KUKA KRL program: MyProgram_129().src

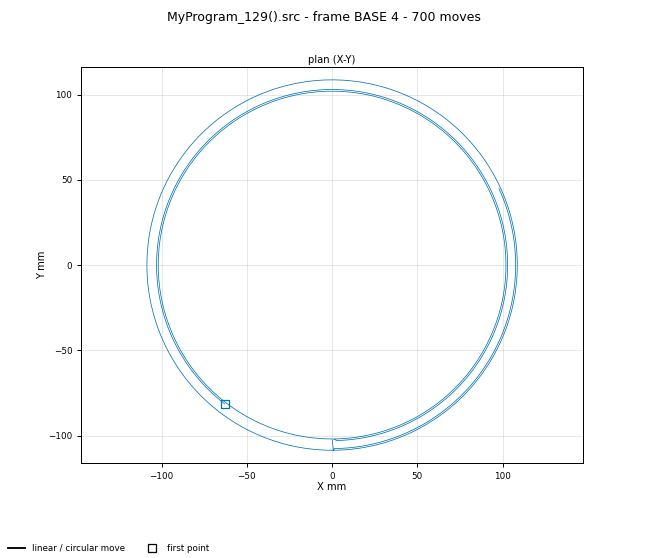
[picture p0: tool path of MyProgram_129().src in frame BASE 4, 700 of 700 moves have a stored position in this frame; points joined in program order, loops and branches not executed]
&ACCESS RVP
&REL 1
&PARAM TEMPLATE = C:\KRC\Roboter\Template\vorgabe
&PARAM EDITMASK = *
DEF MyProgram_129()
; ---- Setting reference (Base) ----
$BASE = BASE_DATA[4]

; --------------------------
; ---- Setting tool (TCP) ----
$TOOL = TOOL_DATA[3]
; --------------------------

$VEL.CP = VEL_APROX_PRINT
Startdeposition()
$VEL.CP = VEL_PRINT
LIN {X -62.9658,Y -81.4453,Z 106,A -132.2913,B 24.9442,C -1.7248,E1 24.9012,E2 217.9169} C_DIS
LIN {X -65.6067,Y -79.3337,Z 106,A -134.1331,B 24.9439,C -1.7297,E1 24.8972,E2 219.7539} C_DIS
LIN {X -68.2811,Y -77.0452,Z 106,A -136.1102,B 24.9437,C -1.7329,E1 24.893,E2 221.7312} C_DIS
LIN {X -70.4655,Y -75.0509,Z 106,A -137.9265,B 24.9439,C -1.7301,E1 24.8893,E2 223.5615} C_DIS
LIN {X -73.3174,Y -72.2675,Z 106,A -139.9622,B 24.9432,C -1.7414,E1 24.8853,E2 225.5791} C_DIS
LIN {X -75.616,Y -69.8596,Z 106,A -142.0598,B 24.9435,C -1.7367,E1 24.8812,E2 227.697} C_DIS
LIN {X -78.3073,Y -66.8281,Z 106,A -144.1543,B 24.9428,C -1.7476,E1 24.8774,E2 229.7748} C_DIS
LIN {X -80.8839,Y -63.6856,Z 106,A -146.4557,B 24.9425,C -1.7516,E1 24.8734,E2 232.0776} C_DIS
LIN {X -82.6713,Y -61.3501,Z 106,A -147.9403,B 24.9419,C -1.7609,E1 24.8709,E2 233.547} C_DIS
LIN {X -84.3493,Y -59.0196,Z 106,A -149.6735,B 24.9419,C -1.7602,E1 24.8681,E2 235.2905} C_DIS
LIN {X -86.3097,Y -56.1161,Z 106,A -151.7179,B 24.9419,C -1.7618,E1 24.8649,E2 237.3412} C_DIS
LIN {X -88.3102,Y -52.9122,Z 106,A -153.6162,B 24.941,C -1.7746,E1 24.8622,E2 239.2189} C_DIS
LIN {X -89.3427,Y -51.1462,Z 106,A -155.0866,B 24.9415,C -1.766,E1 24.8601,E2 240.7174} C_DIS
LIN {X -91.3359,Y -47.498,Z 106,A -157.1631,B 24.9406,C -1.7806,E1 24.8574,E2 242.77} C_DIS
LIN {X -93.0269,Y -44.0942,Z 106,A -159.4092,B 24.9405,C -1.782,E1 24.8547,E2 245.025} C_DIS
LIN {X -94.4755,Y -40.8958,Z 106,A -161.3998,B 24.9402,C -1.7863,E1 24.8524,E2 247.0162} C_DIS
LIN {X -95.9861,Y -37.2142,Z 106,A -163.4255,B 24.9393,C -1.7994,E1 24.8503,E2 249.0222} C_DIS
LIN {X -97.1234,Y -34.133,Z 106,A -165.4942,B 24.9395,C -1.7964,E1 24.8484,E2 251.1096} C_DIS
LIN {X -98.3351,Y -30.4667,Z 106,A -167.5356,B 24.9388,C -1.8066,E1 24.8466,E2 253.1384} C_DIS
LIN {X -99.2194,Y -27.4578,Z 106,A -169.3316,B 24.9386,C -1.8101,E1 24.8453,E2 254.9364} C_DIS
LIN {X -100.529,Y -22.1809,Z 106,A -172.0309,B 24.9372,C -1.8308,E1 24.8435,E2 257.6021} C_DIS
LIN {X -101.1949,Y -18.9188,Z 106,A -174.3718,B 24.9379,C -1.8197,E1 24.8422,E2 259.9835} C_DIS
LIN {X -101.8925,Y -14.6964,Z 106,A -176.5465,B 24.9369,C -1.8344,E1 24.8413,E2 262.136} C_DIS
LIN {X -102.234,Y -12.0934,Z 106,A -178.0467,B 24.9367,C -1.8377,E1 24.8408,E2 263.6374} C_DIS
LIN {X -102.5546,Y -8.9886,Z 106,A -179.9416,B 24.9367,C -1.8377,E1 24.8403,E2 265.5434} C_DIS
LIN {X -102.8206,Y -5.1232,Z 106,A 177.9162,B 24.9362,C -1.8452,E1 24.8399,E2 267.6808} C_DIS
LIN {X -102.9266,Y -2.0367,Z 106,A 176.3907,B 24.9353,C -1.8574,E1 24.8399,E2 269.1864} C_DIS
LIN {X -102.9421,Y 1.0814,Z 106,A 174.6385,B 24.935,C -1.8624,E1 24.8399,E2 270.9372} C_DIS
LIN {X -102.8555,Y 4.3316,Z 106,A 172.9749,B 24.9342,C -1.8733,E1 24.8399,E2 272.5849} C_DIS
LIN {X -102.6601,Y 7.6926,Z 106,A 170.758,B 24.9346,C -1.8675,E1 24.8404,E2 274.8289} C_DIS
LIN {X -102.3213,Y 11.3472,Z 106,A 168.6519,B 24.9343,C -1.8719,E1 24.8409,E2 276.9371} C_DIS
LIN {X -101.8299,Y 15.1348,Z 106,A 166.6862,B 24.9334,C -1.8843,E1 24.8417,E2 278.8851} C_DIS
LIN {X -101.2979,Y 18.3511,Z 106,A 164.7721,B 24.9333,C -1.8867,E1 24.8426,E2 280.8047} C_DIS
LIN {X -100.3856,Y 22.8227,Z 106,A 162.208,B 24.9328,C -1.894,E1 24.8441,E2 283.3665} C_DIS
LIN {X -99.542,Y 26.2634,Z 106,A 160.1806,B 24.9324,C -1.8983,E1 24.8455,E2 285.3955} C_DIS
LIN {X -98.7388,Y 29.1324,Z 106,A 158.4759,B 24.9322,C -1.902,E1 24.8468,E2 287.1013} C_DIS
LIN {X -97.7556,Y 32.2837,Z 106,A 156.7577,B 24.9315,C -1.9118,E1 24.8483,E2 288.8059} C_DIS
LIN {X -96.565,Y 35.6848,Z 106,A 154.8063,B 24.9309,C -1.9199,E1 24.8501,E2 290.7491} C_DIS
LIN {X -95.1884,Y 39.2093,Z 106,A 152.6847,B 24.9305,C -1.9258,E1 24.8523,E2 292.8684} C_DIS
LIN {X -93.4142,Y 43.2647,Z 106,A 150.4424,B 24.9294,C -1.9409,E1 24.8548,E2 295.0869} C_DIS
LIN {X -92.6832,Y 44.8096,Z 106,A 148.8667,B 24.9307,C -1.9222,E1 24.8568,E2 296.7159} C_DIS
LIN {X -90.7079,Y 48.6857,Z 106,A 146.6291,B 24.9298,C -1.9357,E1 24.8596,E2 298.9333} C_DIS
LIN {X -88.9696,Y 51.7954,Z 106,A 144.6192,B 24.9294,C -1.9405,E1 24.8624,E2 300.9422} C_DIS
LIN {X -87.387,Y 54.4202,Z 106,A 142.3126,B 24.9306,C -1.9247,E1 24.8659,E2 303.2983} C_DIS
LIN {X -84.9704,Y 58.1231,Z 106,A 140.4496,B 24.9286,C -1.9521,E1 24.8687,E2 305.1051} C_DIS
LIN {X -82.9524,Y 60.9668,Z 106,A 138.6482,B 24.9278,C -1.9623,E1 24.8716,E2 306.8911} C_DIS
LIN {X -80.8826,Y 63.6871,Z 106,A 136.6902,B 24.9276,C -1.9654,E1 24.875,E2 308.8509} C_DIS
LIN {X -78.8684,Y 66.1667,Z 106,A 134.7875,B 24.9276,C -1.9657,E1 24.8784,E2 310.7617} C_DIS
LIN {X -76.5485,Y 68.836,Z 106,A 132.7968,B 24.9272,C -1.9699,E1 24.8821,E2 312.7512} C_DIS
LIN {X -74.1207,Y 71.4433,Z 106,A 130.8532,B 24.9268,C -1.9762,E1 24.8858,E2 314.6883} C_DIS
LIN {X -71.6032,Y 73.9666,Z 106,A 128.9157,B 24.9263,C -1.9826,E1 24.8896,E2 316.6187} C_DIS
LIN {X -69.7194,Y 75.7447,Z 106,A 127.3147,B 24.9265,C -1.9804,E1 24.8929,E2 318.2315} C_DIS
LIN {X -66.7732,Y 78.3541,Z 106,A 125.2257,B 24.9258,C -1.9889,E1 24.8973,E2 320.3083} C_DIS
LIN {X -63.9199,Y 80.6987,Z 106,A 123.2261,B 24.9253,C -1.9954,E1 24.9016,E2 322.3001} C_DIS
LIN {X -61.0609,Y 82.8835,Z 106,A 121.1752,B 24.9252,C -1.9978,E1 24.9062,E2 324.3525} C_DIS
LIN {X -58.2959,Y 84.8524,Z 106,A 119.194,B 24.9252,C -1.9984,E1 24.9108,E2 326.3392} C_DIS
LIN {X -53.6434,Y 87.8661,Z 106,A 115.5962,B 24.926,C -1.9861,E1 24.9194,E2 329.9777} C_DIS
LIN {X -50.2253,Y 89.8635,Z 106,A 113.9609,B 24.9242,C -2.0101,E1 24.9232,E2 331.5606} C_DIS
LIN {X -48.073,Y 91.0331,Z 106,A 112.0791,B 24.9255,C -1.9939,E1 24.928,E2 333.4861} C_DIS
LIN {X -44.7451,Y 92.7142,Z 106,A 110.4816,B 24.9239,C -2.0143,E1 24.9319,E2 335.0393} C_DIS
LIN {X -41.3,Y 94.2993,Z 106,A 108.358,B 24.9237,C -2.017,E1 24.9373,E2 337.1617} C_DIS
LIN {X -38.1812,Y 95.6062,Z 106,A 106.2801,B 24.9241,C -2.0125,E1 24.9427,E2 339.2548} C_DIS
LIN {X -34.2728,Y 97.0744,Z 106,A 103.6233,B 24.9247,C -2.0035,E1 24.9498,E2 341.9383} C_DIS
LIN {X -30.6042,Y 98.2925,Z 106,A 102.0428,B 24.923,C -2.0267,E1 24.9538,E2 343.4666} C_DIS
LIN {X -27.3929,Y 99.2369,Z 106,A 100.0954,B 24.923,C -2.0255,E1 24.9591,E2 345.4197} C_DIS
LIN {X -24.6455,Y 99.9534,Z 106,A 97.9782,B 24.9244,C -2.0075,E1 24.9649,E2 347.5826} C_DIS
LIN {X -20.7417,Y 100.8355,Z 106,A 96.3511,B 24.9226,C -2.0314,E1 24.9692,E2 349.1551} C_DIS
LIN {X -17.204,Y 101.4992,Z 106,A 94.3488,B 24.9226,C -2.0329,E1 24.9747,E2 351.1558} C_DIS
LIN {X -13.8035,Y 102.0187,Z 106,A 92.2968,B 24.9228,C -2.0291,E1 24.9804,E2 353.2186} C_DIS
LIN {X -9.7729,Y 102.4822,Z 106,A 90.306,B 24.9219,C -2.0402,E1 24.9859,E2 355.1842} C_DIS
LIN {X -7.5868,Y 102.6686,Z 106,A 89.0458,B 24.922,C -2.0393,E1 24.9894,E2 356.4471} C_DIS
LIN {X -5.0186,Y 102.8259,Z 106,A 87.4239,B 24.9225,C -2.0327,E1 24.994,E2 358.085} C_DIS
LIN {X -1.4379,Y 102.9376,Z 106,A 85.4318,B 24.9225,C -2.0333,E1 24.9995,E2 360.0758} C_DIS
LIN {X 2.5172,Y 102.9178,Z 106,A 83.2645,B 24.9224,C -2.0349,E1 25.0056,E2 362.2391} C_DIS
LIN {X 5.7768,Y 102.7845,Z 106,A 81.5245,B 24.9221,C -2.0379,E1 25.0104,E2 363.9716} C_DIS
LIN {X 9.325,Y 102.5236,Z 106,A 79.5382,B 24.9221,C -2.0375,E1 25.0159,E2 365.9577} C_DIS
LIN {X 12.8225,Y 102.1458,Z 106,A 77.6951,B 24.9218,C -2.0415,E1 25.021,E2 367.7899} C_DIS
LIN {X 16.0252,Y 101.6922,Z 106,A 75.6786,B 24.9225,C -2.0328,E1 25.0266,E2 369.8252} C_DIS
LIN {X 19.6144,Y 101.061,Z 106,A 73.6759,B 24.9225,C -2.033,E1 25.0321,E2 371.8253} C_DIS
LIN {X 22.9736,Y 100.3507,Z 106,A 72.0093,B 24.9219,C -2.0414,E1 25.0366,E2 373.4698} C_DIS
LIN {X 27.326,Y 99.255,Z 106,A 69.2422,B 24.9228,C -2.0295,E1 25.0442,E2 376.2608} C_DIS
LIN {X 29.9394,Y 98.4986,Z 106,A 67.65,B 24.9231,C -2.0253,E1 25.0484,E2 377.86} C_DIS
LIN {X 33.8919,Y 97.208,Z 106,A 65.683,B 24.9222,C -2.0368,E1 25.0535,E2 379.7961} C_DIS
LIN {X 36.5797,Y 96.2287,Z 106,A 63.8725,B 24.923,C -2.0268,E1 25.0583,E2 381.6263} C_DIS
LIN {X 39.4197,Y 95.1024,Z 106,A 62.0629,B 24.9234,C -2.0208,E1 25.063,E2 383.4461} C_DIS
LIN {X 41.9663,Y 94.0052,Z 106,A 60.6164,B 24.9233,C -2.0229,E1 25.0667,E2 384.8842} C_DIS
LIN {X 45.5013,Y 92.3456,Z 106,A 58.7162,B 24.9227,C -2.0309,E1 25.0714,E2 386.7604} C_DIS
LIN {X 49.0753,Y 90.4966,Z 106,A 56.2884,B 24.9234,C -2.0205,E1 25.0775,E2 389.2059} C_DIS
LIN {X 52.3872,Y 88.6205,Z 106,A 54.1796,B 24.9237,C -2.0179,E1 25.0826,E2 391.3147} C_DIS
LIN {X 55.5222,Y 86.6909,Z 106,A 52.2641,B 24.9235,C -2.02,E1 25.0871,E2 393.2191} C_DIS
LIN {X 58.6075,Y 84.6358,Z 106,A 50.0537,B 24.9242,C -2.0108,E1 25.0923,E2 395.4438} C_DIS
LIN {X 61.4156,Y 82.6221,Z 106,A 47.9904,B 24.9249,C -2.0018,E1 25.0969,E2 397.5208} C_DIS
LIN {X 64.588,Y 80.1655,Z 106,A 45.9882,B 24.9245,C -2.0069,E1 25.1013,E2 399.5037} C_DIS
LIN {X 66.6939,Y 78.4216,Z 106,A 44.4814,B 24.9247,C -2.0046,E1 25.1045,E2 401.0102} C_DIS
LIN {X 70.9764,Y 74.5704,Z 106,A 41.121,B 24.9256,C -1.9918,E1 25.1115,E2 404.387} C_DIS
LIN {X 74.6601,Y 70.8811,Z 106,A 38.2942,B 24.9259,C -1.9886,E1 25.117,E2 407.2095} C_DIS
LIN {X 77.0634,Y 68.2608,Z 106,A 36.3087,B 24.9262,C -1.9838,E1 25.1207,E2 409.1974} C_DIS
LIN {X 79.1319,Y 65.8496,Z 106,A 34.6241,B 24.9262,C -1.9831,E1 25.1237,E2 410.8761} C_DIS
LIN {X 81.6934,Y 62.644,Z 106,A 32.3281,B 24.9267,C -1.9771,E1 25.1277,E2 413.1755} C_DIS
LIN {X 83.7613,Y 59.8504,Z 106,A 30.7349,B 24.926,C -1.9861,E1 25.1303,E2 414.7397} C_DIS
LIN {X 85.3156,Y 57.6132,Z 106,A 28.9379,B 24.9272,C -1.9708,E1 25.1332,E2 416.564} C_DIS
LIN {X 87.1419,Y 54.8124,Z 106,A 27.0175,B 24.9277,C -1.9635,E1 25.1361,E2 418.4919} C_DIS
LIN {X 89.0218,Y 51.7045,Z 106,A 24.8036,B 24.9287,C -1.9503,E1 25.1392,E2 420.7257} C_DIS
LIN {X 90.8591,Y 48.4033,Z 106,A 23.0909,B 24.9279,C -1.9604,E1 25.1415,E2 422.4055} C_DIS
LIN {X 92.2425,Y 45.7093,Z 106,A 21.3274,B 24.9285,C -1.9526,E1 25.1437,E2 424.1782} C_DIS
LIN {X 93.7869,Y 42.4506,Z 106,A 19.2787,B 24.9291,C -1.9451,E1 25.1461,E2 426.2333} C_DIS
LIN {X 95.2034,Y 39.1726,Z 106,A 17.266,B 24.9296,C -1.9383,E1 25.1483,E2 428.251} C_DIS
LIN {X 96.1225,Y 36.8598,Z 106,A 15.8165,B 24.93,C -1.9316,E1 25.1498,E2 429.7083} C_DIS
LIN {X 97.8586,Y 31.9654,Z 106,A 12.7411,B 24.9312,C -1.9154,E1 25.1526,E2 432.8046} C_DIS
LIN {X 99.2314,Y 27.4134,Z 106,A 10.2897,B 24.9312,C -1.9154,E1 25.1545,E2 435.2422} C_DIS
LIN {X 100.1851,Y 23.6907,Z 106,A 8.3571,B 24.9311,C -1.9172,E1 25.1558,E2 437.1592} C_DIS
LIN {X 100.7168,Y 21.3202,Z 106,A 6.8767,B 24.9318,C -1.9077,E1 25.1566,E2 438.6534} C_DIS
LIN {X 101.4653,Y 17.407,Z 106,A 4.6703,B 24.9322,C -1.9012,E1 25.1577,E2 440.8622} C_DIS
LIN {X 102.038,Y 13.6544,Z 106,A 2.8259,B 24.9319,C -1.9056,E1 25.1585,E2 442.6854} C_DIS
LIN {X 102.3891,Y 10.6999,Z 106,A 1.2723,B 24.9319,C -1.9046,E1 25.159,E2 444.2322} C_DIS
LIN {X 102.6225,Y 8.1632,Z 106,A -0.3648,B 24.933,C -1.8909,E1 25.1594,E2 445.8918} C_DIS
LIN {X 102.8581,Y 4.2729,Z 106,A -2.4918,B 24.9333,C -1.8857,E1 25.1597,E2 448.0184} C_DIS
LIN {X 102.9433,Y 0.8921,Z 106,A -4.4678,B 24.934,C -1.8757,E1 25.1597,E2 450.0062} C_DIS
LIN {X 102.898,Y -3.166,Z 106,A -6.5956,B 24.9342,C -1.8739,E1 25.1597,E2 452.1258} C_DIS
LIN {X 102.7469,Y -6.4315,Z 106,A -8.5187,B 24.9349,C -1.8636,E1 25.1594,E2 454.0615} C_DIS
LIN {X 102.4581,Y -10.0339,Z 106,A -10.5904,B 24.9355,C -1.8546,E1 25.1589,E2 456.1422} C_DIS
LIN {X 102.0263,Y -13.7451,Z 106,A -12.6743,B 24.936,C -1.8477,E1 25.1581,E2 458.2301} C_DIS
LIN {X 101.4114,Y -17.72,Z 106,A -14.815,B 24.9362,C -1.8445,E1 25.1572,E2 460.3657} C_DIS
LIN {X 100.7451,Y -21.182,Z 106,A -16.5807,B 24.9361,C -1.8464,E1 25.1562,E2 462.1167} C_DIS
LIN {X 99.424,Y -26.7004,Z 106,A -19.8891,B 24.9372,C -1.8301,E1 25.154,E2 465.4445} C_DIS
LIN {X 98.6154,Y -29.5483,Z 106,A -21.9381,B 24.9387,C -1.8083,E1 25.1523,E2 467.5332} C_DIS
LIN {X 97.5583,Y -32.8694,Z 106,A -23.3998,B 24.9378,C -1.8219,E1 25.1511,E2 468.9545} C_DIS
LIN {X 96.556,Y -35.7095,Z 106,A -25.3725,B 24.939,C -1.8044,E1 25.1491,E2 470.9573} C_DIS
LIN {X 94.7059,Y -40.3607,Z 106,A -27.7327,B 24.9384,C -1.8135,E1 25.1467,E2 473.2833} C_DIS
LIN {X 93.478,Y -43.1277,Z 106,A -29.4952,B 24.9389,C -1.8051,E1 25.1446,E2 475.0559} C_DIS
LIN {X 92.1175,Y -45.9614,Z 106,A -31.5531,B 24.9401,C -1.7872,E1 25.1421,E2 477.1451} C_DIS
LIN {X 89.8968,Y -50.1655,Z 106,A -33.8491,B 24.9397,C -1.7938,E1 25.139,E2 479.4134} C_DIS
LIN {X 88.2312,Y -53.0426,Z 106,A -35.5396,B 24.9397,C -1.795,E1 25.1367,E2 481.0925} C_DIS
LIN {X 86.6142,Y -55.6417,Z 106,A -37.4247,B 24.9404,C -1.7827,E1 25.1338,E2 482.9971} C_DIS
LIN {X 84.4817,Y -58.8291,Z 106,A -39.4241,B 24.9404,C -1.7822,E1 25.1307,E2 484.9876} C_DIS
LIN {X 82.62,Y -61.4184,Z 106,A -41.3444,B 24.9412,C -1.7714,E1 25.1275,E2 486.9243} C_DIS
LIN {X 80.5085,Y -64.1605,Z 106,A -43.259,B 24.9415,C -1.7667,E1 25.1242,E2 488.841} C_DIS
LIN {X 77.9596,Y -67.2362,Z 106,A -45.4651,B 24.9418,C -1.7615,E1 25.1202,E2 491.0491} C_DIS
LIN {X 75.2252,Y -70.2801,Z 106,A -47.7079,B 24.9421,C -1.7572,E1 25.116,E2 493.2924} C_DIS
LIN {X 72.6517,Y -72.9379,Z 106,A -49.7736,B 24.9425,C -1.7518,E1 25.112,E2 495.3619} C_DIS
LIN {X 70.1893,Y -75.3107,Z 106,A -51.6862,B 24.9428,C -1.7469,E1 25.1081,E2 497.2783} C_DIS
LIN {X 67.2974,Y -77.9063,Z 106,A -53.8377,B 24.9431,C -1.7424,E1 25.1036,E2 499.4319} C_DIS
LIN {X 64.6832,Y -80.0883,Z 106,A -55.7071,B 24.9433,C -1.7392,E1 25.0995,E2 501.3016} C_DIS
LIN {X 61.7869,Y -82.3432,Z 106,A -57.6613,B 24.9433,C -1.7384,E1 25.0952,E2 503.2506} C_DIS
LIN {X 59.2069,Y -84.2191,Z 106,A -59.3837,B 24.9435,C -1.7369,E1 25.0913,E2 504.9706} C_DIS
LIN {X 56.455,Y -86.0867,Z 106,A -61.3494,B 24.944,C -1.7286,E1 25.0867,E2 506.9493} C_DIS
LIN {X 54.0042,Y -87.6468,Z 106,A -63.0553,B 24.9444,C -1.7219,E1 25.0826,E2 508.6657} C_DIS
LIN {X 50.51,Y -89.7045,Z 106,A -65.0785,B 24.9441,C -1.7272,E1 25.0778,E2 510.6703} C_DIS
LIN {X 47.2158,Y -91.4815,Z 106,A -67.2395,B 24.9445,C -1.7205,E1 25.0724,E2 512.8409} C_DIS
LIN {X 44.5487,Y -92.8086,Z 106,A -69.2066,B 24.9455,C -1.7055,E1 25.0674,E2 514.8383} C_DIS
LIN {X 40.1103,Y -94.8114,Z 106,A -71.6113,B 24.945,C -1.7135,E1 25.0613,E2 517.2181} C_DIS
LIN {X 36.8887,Y -96.1117,Z 106,A -73.329,B 24.9446,C -1.7194,E1 25.0569,E2 518.9182} C_DIS
LIN {X 32.1364,Y -97.8033,Z 106,A -76.3062,B 24.9453,C -1.709,E1 25.049,E2 521.914} C_DIS
LIN {X 29.3754,Y -98.6667,Z 106,A -78.6501,B 24.9472,C -1.6784,E1 25.0426,E2 524.3262} C_DIS
LIN {X 24.9574,Y -99.8773,Z 106,A -80.5539,B 24.9458,C -1.701,E1 25.0376,E2 526.1737} C_DIS
LIN {X 21.2422,Y -100.7328,Z 106,A -82.6531,B 24.9458,C -1.6999,E1 25.0318,E2 528.2726} C_DIS
LIN {X 18.1813,Y -101.3285,Z 106,A -84.3476,B 24.9458,C -1.7001,E1 25.0272,E2 529.9647} C_DIS
LIN {X 14.0786,Y -101.9803,Z 106,A -86.8114,B 24.9463,C -1.6926,E1 25.0204,E2 532.4441} C_DIS
LIN {X 9.9325,Y -102.4675,Z 106,A -89.0321,B 24.9461,C -1.6952,E1 25.0142,E2 534.6571} C_DIS
LIN {X 6.1406,Y -102.7644,Z 106,A -90.9312,B 24.9457,C -1.7027,E1 25.009,E2 536.5376} C_DIS
LIN {X 2.8466,Y -102.9078,Z 106,A -92.931,B 24.9461,C -1.6957,E1 25.0033,E2 538.5535} C_DIS
LIN {X 2.8466,Y -102.9078,Z 106,A -92.931,B 24.9461,C -1.6957,E1 25.0033,E2 538.5535} C_DIS
Enddeposition()
LIN {X 0.7303,Y -101.9715,Z 106,A -93.7462,B 24.9441,C -1.7264,E1 25.0013,E2 539.2958} C_DIS
Startdeposition()
$VEL.CP = VEL_PRINT
LIN {X 3.7248,Y -101.9078,Z 106,A -91.6833,B 24.9432,C -1.7415,E1 25.0071,E2 537.1974} C_DIS
LIN {X 6.2515,Y -101.7842,Z 106,A -90.2592,B 24.9432,C -1.7422,E1 25.0111,E2 535.7723} C_DIS
LIN {X 8.5664,Y -101.6146,Z 106,A -88.9449,B 24.943,C -1.7432,E1 25.0148,E2 534.4561} C_DIS
LIN {X 11.2257,Y -101.3562,Z 106,A -87.3849,B 24.9428,C -1.7464,E1 25.0191,E2 532.8897} C_DIS
LIN {X 14.3772,Y -100.9555,Z 106,A -85.5987,B 24.9428,C -1.7476,E1 25.0241,E2 531.1021} C_DIS
LIN {X 17.431,Y -100.4752,Z 106,A -83.9407,B 24.9428,C -1.7458,E1 25.0286,E2 529.45} C_DIS
LIN {X 19.887,Y -100.018,Z 106,A -82.5398,B 24.9428,C -1.7469,E1 25.0325,E2 528.0482} C_DIS
LIN {X 22.1593,Y -99.5383,Z 106,A -81.2252,B 24.9428,C -1.7485,E1 25.0361,E2 526.7316} C_DIS
LIN {X 24.573,Y -98.97,Z 106,A -79.8007,B 24.9425,C -1.7511,E1 25.0399,E2 525.3029} C_DIS
LIN {X 27.9046,Y -98.0819,Z 106,A -77.832,B 24.9423,C -1.7544,E1 25.0452,E2 523.3295} C_DIS
LIN {X 31.443,Y -97.0054,Z 106,A -75.7728,B 24.9422,C -1.7561,E1 25.0507,E2 521.27} C_DIS
LIN {X 34.326,Y -96.025,Z 106,A -74.1374,B 24.9422,C -1.7553,E1 25.055,E2 519.6398} C_DIS
LIN {X 36.5361,Y -95.2052,Z 106,A -72.8033,B 24.9422,C -1.7575,E1 25.0585,E2 518.3034} C_DIS
LIN {X 38.8533,Y -94.2832,Z 106,A -71.4058,B 24.942,C -1.7593,E1 25.0621,E2 516.9048} C_DIS
LIN {X 41.1468,Y -93.3051,Z 106,A -70.009,B 24.9419,C -1.7613,E1 25.0657,E2 515.5067} C_DIS
LIN {X 43.5274,Y -92.2192,Z 106,A -68.554,B 24.9417,C -1.763,E1 25.0694,E2 514.0514} C_DIS
LIN {X 45.6455,Y -91.1886,Z 106,A -67.2326,B 24.9417,C -1.7651,E1 25.0727,E2 512.7286} C_DIS
LIN {X 47.7355,Y -90.1115,Z 106,A -65.8924,B 24.9414,C -1.7681,E1 25.076,E2 511.3849} C_DIS
LIN {X 50.1171,Y -88.8099,Z 106,A -64.3889,B 24.9413,C -1.7699,E1 25.0797,E2 509.8815} C_DIS
LIN {X 52.4282,Y -87.4665,Z 106,A -62.9066,B 24.9412,C -1.7719,E1 25.0833,E2 508.3992} C_DIS
LIN {X 54.5548,Y -86.1561,Z 106,A -61.5087,B 24.941,C -1.7744,E1 25.0866,E2 506.9999} C_DIS
LIN {X 57.6827,Y -84.094,Z 106,A -59.4126,B 24.9407,C -1.7782,E1 25.0915,E2 504.9018} C_DIS
LIN {X 59.658,Y -82.7037,Z 106,A -58.054,B 24.9405,C -1.781,E1 25.0946,E2 503.5412} C_DIS
LIN {X 62.1739,Y -80.8277,Z 106,A -56.2822,B 24.9403,C -1.7852,E1 25.0985,E2 501.766} C_DIS
LIN {X 64.6181,Y -78.8891,Z 106,A -54.5578,B 24.9401,C -1.7879,E1 25.1023,E2 500.0417} C_DIS
LIN {X 67.0013,Y -76.8736,Z 106,A -52.7705,B 24.9397,C -1.7932,E1 25.1061,E2 498.2488} C_DIS
LIN {X 69.473,Y -74.6491,Z 106,A -50.7799,B 24.9391,C -1.8026,E1 25.1102,E2 496.244} C_DIS
LIN {X 72.0408,Y -72.1742,Z 106,A -48.7671,B 24.9387,C -1.8078,E1 25.1142,E2 494.2274} C_DIS
LIN {X 74.2744,Y -69.8715,Z 106,A -47.0625,B 24.9387,C -1.8084,E1 25.1175,E2 492.5289} C_DIS
LIN {X 76.7287,Y -67.1671,Z 106,A -45.0971,B 24.9386,C -1.8101,E1 25.1211,E2 490.5683} C_DIS
LIN {X 78.7706,Y -64.7625,Z 106,A -43.1703,B 24.9378,C -1.821,E1 25.1246,E2 488.6244} C_DIS
LIN {X 80.7685,Y -62.2508,Z 106,A -41.4896,B 24.9378,C -1.8209,E1 25.1275,E2 486.9521} C_DIS
LIN {X 82.5308,Y -59.8963,Z 106,A -39.9322,B 24.9378,C -1.8215,E1 25.13,E2 485.4007} C_DIS
LIN {X 84.0893,Y -57.6896,Z 106,A -38.4239,B 24.9376,C -1.8253,E1 25.1325,E2 483.8908} C_DIS
LIN {X 85.4772,Y -55.6125,Z 106,A -37.0281,B 24.9373,C -1.8289,E1 25.1346,E2 482.4933} C_DIS
LIN {X 86.7207,Y -53.6511,Z 106,A -35.7314,B 24.9371,C -1.8323,E1 25.1365,E2 481.1952} C_DIS
LIN {X 88.0087,Y -51.511,Z 106,A -34.3767,B 24.9369,C -1.8344,E1 25.1384,E2 479.8426} C_DIS
LIN {X 89.3381,Y -49.1712,Z 106,A -32.8338,B 24.9365,C -1.8401,E1 25.1406,E2 478.2943} C_DIS
LIN {X 90.4481,Y -47.0964,Z 106,A -31.5022,B 24.9362,C -1.8444,E1 25.1423,E2 476.9595} C_DIS
LIN {X 91.6499,Y -44.7144,Z 106,A -30.0391,B 24.936,C -1.8474,E1 25.1441,E2 475.4971} C_DIS
LIN {X 92.6423,Y -42.6184,Z 106,A -28.7366,B 24.9358,C -1.8513,E1 25.1457,E2 474.1925} C_DIS
LIN {X 93.7271,Y -40.1788,Z 106,A -27.2462,B 24.9355,C -1.8555,E1 25.1473,E2 472.7004} C_DIS
LIN {X 94.6818,Y -37.874,Z 106,A -25.8545,B 24.9352,C -1.8594,E1 25.1488,E2 471.3072} C_DIS
LIN {X 95.5652,Y -35.5855,Z 106,A -24.4834,B 24.9349,C -1.8634,E1 25.1501,E2 469.9343} C_DIS
LIN {X 96.3676,Y -33.3495,Z 106,A -23.1478,B 24.9346,C -1.8676,E1 25.1514,E2 468.5962} C_DIS
LIN {X 97.2053,Y -30.8252,Z 106,A -21.6749,B 24.9344,C -1.8714,E1 25.1527,E2 467.1227} C_DIS
LIN {X 97.8404,Y -28.741,Z 106,A -20.426,B 24.934,C -1.8763,E1 25.1536,E2 465.8693} C_DIS
LIN {X 98.5273,Y -26.2902,Z 106,A -19.0314,B 24.9338,C -1.8794,E1 25.1547,E2 464.4756} C_DIS
LIN {X 99.1038,Y -24.0242,Z 106,A -17.6652,B 24.9333,C -1.8857,E1 25.1556,E2 463.1022} C_DIS
LIN {X 99.7652,Y -21.119,Z 106,A -16.0721,B 24.9332,C -1.8877,E1 25.1565,E2 461.5136} C_DIS
LIN {X 100.4741,Y -17.437,Z 106,A -13.9793,B 24.9328,C -1.8939,E1 25.1576,E2 459.4185} C_DIS
LIN {X 100.8711,Y -14.9705,Z 106,A -12.5857,B 24.9325,C -1.898,E1 25.1582,E2 458.0234} C_DIS
LIN {X 101.1875,Y -12.6499,Z 106,A -11.2663,B 24.9322,C -1.9024,E1 25.1587,E2 456.7014} C_DIS
LIN {X 101.4667,Y -10.1694,Z 106,A -9.89,B 24.9319,C -1.9059,E1 25.1591,E2 455.3251} C_DIS
LIN {X 101.6992,Y -7.5077,Z 106,A -8.395,B 24.9316,C -1.9105,E1 25.1594,E2 453.8281} C_DIS
LIN {X 101.8428,Y -5.1916,Z 106,A -7.0887,B 24.9313,C -1.9148,E1 25.1596,E2 452.5194} C_DIS
LIN {X 101.9393,Y -2.698,Z 106,A -5.7059,B 24.931,C -1.9186,E1 25.1598,E2 451.136} C_DIS
LIN {X 101.9758,Y 0.0026,Z 106,A -4.2199,B 24.9307,C -1.9221,E1 25.1598,E2 449.6504} C_DIS
LIN {X 101.9454,Y 2.4962,Z 106,A -2.8096,B 24.9304,C -1.927,E1 25.1598,E2 448.2369} C_DIS
LIN {X 101.8614,Y 4.8128,Z 106,A -1.5045,B 24.9301,C -1.9314,E1 25.1596,E2 446.9294} C_DIS
LIN {X 101.7117,Y 7.3249,Z 106,A -0.1121,B 24.9298,C -1.935,E1 25.1593,E2 445.5367} C_DIS
LIN {X 101.4843,Y 10.0016,Z 106,A 1.3854,B 24.9295,C -1.9393,E1 25.1589,E2 444.0377} C_DIS
LIN {X 101.2294,Y 12.3093,Z 106,A 2.6934,B 24.9292,C -1.9437,E1 25.1585,E2 442.7273} C_DIS
LIN {X 100.8729,Y 14.9582,Z 106,A 4.1737,B 24.9289,C -1.9475,E1 25.1579,E2 441.2467} C_DIS
LIN {X 100.4764,Y 17.4237,Z 106,A 5.5667,B 24.9286,C -1.9515,E1 25.1573,E2 439.8524} C_DIS
LIN {X 99.7999,Y 20.9498,Z 106,A 7.5712,B 24.9282,C -1.9573,E1 25.1562,E2 437.8459} C_DIS
LIN {X 99.338,Y 23.0365,Z 106,A 8.8256,B 24.9277,C -1.9633,E1 25.1554,E2 436.5848} C_DIS
LIN {X 98.6539,Y 25.8131,Z 106,A 10.3714,B 24.9276,C -1.9657,E1 25.1543,E2 435.0421} C_DIS
LIN {X 97.7464,Y 29.0579,Z 106,A 12.3001,B 24.927,C -1.9729,E1 25.1528,E2 433.1074} C_DIS
LIN {X 96.9234,Y 31.6965,Z 106,A 13.7715,B 24.927,C -1.9743,E1 25.1516,E2 431.6413} C_DIS
LIN {X 96.151,Y 33.9667,Z 106,A 15.1734,B 24.9265,C -1.9805,E1 25.1503,E2 430.2325} C_DIS
LIN {X 95.2026,Y 36.5429,Z 106,A 16.6296,B 24.9264,C -1.9815,E1 25.1489,E2 428.782} C_DIS
LIN {X 94.2801,Y 38.8609,Z 106,A 18.059,B 24.926,C -1.9867,E1 25.1474,E2 427.3482} C_DIS
LIN {X 93.3012,Y 41.1557,Z 106,A 19.4525,B 24.9257,C -1.9904,E1 25.1458,E2 425.9535} C_DIS
LIN {X 92.1926,Y 43.5845,Z 106,A 20.9301,B 24.9255,C -1.9938,E1 25.1441,E2 424.476} C_DIS
LIN {X 91.2811,Y 45.4589,Z 106,A 22.1344,B 24.9251,C -1.9984,E1 25.1426,E2 423.2672} C_DIS
LIN {X 89.9355,Y 48.0699,Z 106,A 23.7364,B 24.9249,C -2.001,E1 25.1405,E2 421.6676} C_DIS
LIN {X 88.1002,Y 51.3561,Z 106,A 25.8371,B 24.9245,C -2.0061,E1 25.1376,E2 419.5656} C_DIS
LIN {X 86.1565,Y 54.5542,Z 106,A 27.93,B 24.9241,C -2.0113,E1 25.1345,E2 417.4713} C_DIS
LIN {X 84.8925,Y 56.4992,Z 106,A 29.2374,B 24.9239,C -2.0148,E1 25.1325,E2 416.162} C_DIS
LIN {X 83.4852,Y 58.5587,Z 106,A 30.5989,B 24.9237,C -2.0168,E1 25.1304,E2 414.8026} C_DIS
LIN {X 81.9087,Y 60.7459,Z 106,A 32.1265,B 24.9234,C -2.0211,E1 25.1278,E2 413.2723} C_DIS
LIN {X 80.4487,Y 62.6658,Z 106,A 33.6759,B 24.9226,C -2.0322,E1 25.1252,E2 411.7038} C_DIS
LIN {X 78.4255,Y 65.1778,Z 106,A 35.3726,B 24.9226,C -2.0319,E1 25.1222,E2 410.0157} C_DIS
LIN {X 76.3959,Y 67.5482,Z 106,A 37.2134,B 24.922,C -2.0394,E1 25.1188,E2 408.1654} C_DIS
LIN {X 74.2913,Y 69.8535,Z 106,A 38.7881,B 24.9223,C -2.0361,E1 25.1158,E2 406.6055} C_DIS
LIN {X 72.0427,Y 72.1723,Z 106,A 40.7506,B 24.9215,C -2.0459,E1 25.1119,E2 404.628} C_DIS
LIN {X 69.4823,Y 74.6404,Z 106,A 42.7567,B 24.9212,C -2.0504,E1 25.1079,E2 402.6197} C_DIS
LIN {X 67.0104,Y 76.8656,Z 106,A 44.5386,B 24.9212,C -2.0507,E1 25.1041,E2 400.8442} C_DIS
LIN {X 64.2104,Y 79.2196,Z 106,A 46.5674,B 24.9209,C -2.0535,E1 25.0998,E2 398.8165} C_DIS
LIN {X 61.4819,Y 81.3559,Z 106,A 48.5116,B 24.9207,C -2.0569,E1 25.0955,E2 396.8714} C_DIS
LIN {X 59.1858,Y 83.0407,Z 106,A 50.0966,B 24.9205,C -2.0591,E1 25.0919,E2 395.2869} C_DIS
LIN {X 56.88,Y 84.6374,Z 106,A 51.6033,B 24.9205,C -2.0589,E1 25.0884,E2 393.7856} C_DIS
LIN {X 54.701,Y 86.0623,Z 106,A 53.0324,B 24.9205,C -2.0599,E1 25.0851,E2 392.3588} C_DIS
LIN {X 52.5778,Y 87.3756,Z 106,A 54.4305,B 24.9203,C -2.0618,E1 25.0817,E2 390.9605} C_DIS
LIN {X 50.4231,Y 88.6364,Z 106,A 55.8406,B 24.9201,C -2.0642,E1 25.0783,E2 389.5492} C_DIS
LIN {X 48.0822,Y 89.9288,Z 106,A 57.3258,B 24.92,C -2.0655,E1 25.0747,E2 388.065} C_DIS
LIN {X 45.9031,Y 91.0601,Z 106,A 58.6926,B 24.9199,C -2.0668,E1 25.0713,E2 386.6989} C_DIS
LIN {X 43.765,Y 92.1061,Z 106,A 60.0365,B 24.9197,C -2.0687,E1 25.0679,E2 385.3541} C_DIS
LIN {X 41.7298,Y 93.045,Z 106,A 61.3544,B 24.9195,C -2.0725,E1 25.0645,E2 384.0306} C_DIS
LIN {X 39.1852,Y 94.1458,Z 106,A 62.8577,B 24.9195,C -2.072,E1 25.0607,E2 382.5319} C_DIS
LIN {X 36.8684,Y 95.077,Z 106,A 64.258,B 24.9194,C -2.0733,E1 25.057,E2 381.1316} C_DIS
LIN {X 34.3648,Y 96.0112,Z 106,A 65.7443,B 24.9194,C -2.0741,E1 25.0532,E2 379.6466} C_DIS
LIN {X 32.0043,Y 96.8236,Z 106,A 67.1454,B 24.9192,C -2.0752,E1 25.0494,E2 378.2456} C_DIS
LIN {X 28.574,Y 97.8899,Z 106,A 69.1712,B 24.9191,C -2.077,E1 25.044,E2 376.219} C_DIS
LIN {X 26.1786,Y 98.5575,Z 106,A 70.5673,B 24.9191,C -2.0779,E1 25.0403,E2 374.8231} C_DIS
LIN {X 23.5999,Y 99.2074,Z 106,A 72.0455,B 24.9191,C -2.0781,E1 25.0363,E2 373.3465} C_DIS
LIN {X 21.124,Y 99.7641,Z 106,A 73.472,B 24.919,C -2.0789,E1 25.0324,E2 371.9201} C_DIS
LIN {X 18.0768,Y 100.3591,Z 106,A 75.2623,B 24.9188,C -2.0814,E1 25.0274,E2 370.126} C_DIS
LIN {X 14.9608,Y 100.8726,Z 106,A 76.9874,B 24.9188,C -2.08,E1 25.0227,E2 368.4058} C_DIS
LIN {X 12.6594,Y 101.1862,Z 106,A 78.304,B 24.9188,C -2.0807,E1 25.0191,E2 367.0884} C_DIS
LIN {X 10.1768,Y 101.466,Z 106,A 79.696,B 24.9188,C -2.0805,E1 25.0152,E2 365.698} C_DIS
LIN {X 7.5125,Y 101.6988,Z 106,A 81.1988,B 24.9188,C -2.0805,E1 25.011,E2 364.1958} C_DIS
LIN {X 5.185,Y 101.8431,Z 106,A 82.523,B 24.9188,C -2.0811,E1 25.0073,E2 362.8708} C_DIS
LIN {X 2.6766,Y 101.9399,Z 106,A 83.9194,B 24.9188,C -2.0805,E1 25.0034,E2 361.4763} C_DIS
LIN {X 0.0046,Y 101.976,Z 106,A 85.4212,B 24.9188,C -2.0802,E1 24.9992,E2 359.9752} C_DIS
LIN {X -2.4648,Y 101.946,Z 106,A 86.8104,B 24.9188,C -2.0799,E1 24.9954,E2 358.5866} C_DIS
LIN {X -4.8109,Y 101.8614,Z 106,A 88.1421,B 24.9188,C -2.0799,E1 24.9916,E2 357.2546} C_DIS
LIN {X -7.3018,Y 101.7132,Z 106,A 89.5354,B 24.9189,C -2.0791,E1 24.9878,E2 355.8628} C_DIS
LIN {X -9.9922,Y 101.4853,Z 106,A 91.052,B 24.919,C -2.0783,E1 24.9835,E2 354.3473} C_DIS
LIN {X -12.3004,Y 101.2305,Z 106,A 92.3701,B 24.919,C -2.0781,E1 24.9799,E2 353.0289} C_DIS
LIN {X -15.2301,Y 100.831,Z 106,A 94.1358,B 24.9188,C -2.0809,E1 24.975,E2 351.2551} C_DIS
LIN {X -18.4913,Y 100.2845,Z 106,A 95.8944,B 24.9192,C -2.0758,E1 24.9702,E2 349.5068} C_DIS
LIN {X -20.9439,Y 99.8011,Z 106,A 97.2818,B 24.9193,C -2.074,E1 24.9664,E2 348.1221} C_DIS
LIN {X -23.5819,Y 99.2118,Z 106,A 98.8017,B 24.9194,C -2.0726,E1 24.9623,E2 346.6034} C_DIS
LIN {X -25.8267,Y 98.6504,Z 106,A 100.1232,B 24.9194,C -2.0721,E1 24.9587,E2 345.2812} C_DIS
LIN {X -28.227,Y 97.9905,Z 106,A 101.5282,B 24.9196,C -2.0709,E1 24.9549,E2 343.8769} C_DIS
LIN {X -30.5709,Y 97.2845,Z 106,A 102.8989,B 24.9197,C -2.0692,E1 24.9513,E2 342.5079} C_DIS
LIN {X -33.3021,Y 96.3842,Z 106,A 104.682,B 24.9194,C -2.0733,E1 24.9465,E2 340.7117} C_DIS
LIN {X -36.5249,Y 95.2094,Z 106,A 106.4394,B 24.9201,C -2.0646,E1 24.942,E2 338.9714} C_DIS
LIN {X -38.8612,Y 94.28,Z 106,A 107.877,B 24.9201,C -2.0635,E1 24.9382,E2 337.5331} C_DIS
LIN {X -41.1584,Y 93.3,Z 106,A 109.2485,B 24.9204,C -2.0603,E1 24.9347,E2 336.166} C_DIS
LIN {X -43.5899,Y 92.1901,Z 106,A 110.7807,B 24.9204,C -2.0591,E1 24.9308,E2 334.6328} C_DIS
LIN {X -45.5334,Y 91.2442,Z 106,A 112.0234,B 24.9206,C -2.0582,E1 24.9277,E2 333.389} C_DIS
LIN {X -48.0737,Y 89.9334,Z 106,A 113.6097,B 24.9208,C -2.0548,E1 24.9238,E2 331.8065} C_DIS
LIN {X -50.0965,Y 88.8214,Z 106,A 114.9246,B 24.921,C -2.0532,E1 24.9206,E2 330.4916} C_DIS
LIN {X -52.3924,Y 87.4877,Z 106,A 116.4108,B 24.9212,C -2.0502,E1 24.917,E2 329.0078} C_DIS
LIN {X -54.4995,Y 86.1906,Z 106,A 117.8063,B 24.9214,C -2.0478,E1 24.9137,E2 327.6137} C_DIS
LIN {X -56.4165,Y 84.9471,Z 106,A 119.0645,B 24.9216,C -2.0444,E1 24.9108,E2 326.3594} C_DIS
LIN {X -58.2606,Y 83.6924,Z 106,A 120.4476,B 24.9215,C -2.0466,E1 24.9076,E2 324.9665} C_DIS
LIN {X -60.7525,Y 81.9038,Z 106,A 122.279,B 24.9215,C -2.0469,E1 24.9035,E2 323.128} C_DIS
LIN {X -63.3,Y 79.9489,Z 106,A 124.0207,B 24.9219,C -2.0408,E1 24.8997,E2 321.3944} C_DIS
LIN {X -66.1282,Y 77.6259,Z 106,A 125.9864,B 24.9225,C -2.033,E1 24.8955,E2 319.4396} C_DIS
LIN {X -68.4754,Y 75.5659,Z 106,A 127.774,B 24.9227,C -2.0301,E1 24.8917,E2 317.6519} C_DIS
LIN {X -70.7684,Y 73.4203,Z 106,A 129.5992,B 24.9229,C -2.0281,E1 24.888,E2 315.8238} C_DIS
LIN {X -73.358,Y 70.8331,Z 106,A 131.5942,B 24.9234,C -2.0209,E1 24.8841,E2 313.8375} C_DIS
LIN {X -75.2631,Y 68.8056,Z 106,A 133.2841,B 24.9234,C -2.0215,E1 24.8809,E2 312.1389} C_DIS
LIN {X -77.6247,Y 66.1296,Z 106,A 135.2555,B 24.9239,C -2.0152,E1 24.8773,E2 310.1736} C_DIS
LIN {X -79.9482,Y 63.3009,Z 106,A 137.2514,B 24.9244,C -2.0076,E1 24.8738,E2 308.1865} C_DIS
LIN {X -81.7969,Y 60.8948,Z 106,A 138.9423,B 24.9248,C -2.0025,E1 24.871,E2 306.4996} C_DIS
LIN {X -83.0593,Y 59.1598,Z 106,A 140.2409,B 24.9248,C -2.0025,E1 24.8689,E2 305.1947} C_DIS
LIN {X -84.5752,Y 56.972,Z 106,A 141.7225,B 24.9252,C -1.9978,E1 24.8665,E2 303.7169} C_DIS
LIN {X -86.075,Y 54.6812,Z 106,A 143.2076,B 24.9256,C -1.9916,E1 24.8643,E2 302.2391} C_DIS
LIN {X -87.3843,Y 52.5634,Z 106,A 144.6153,B 24.9259,C -1.9879,E1 24.8623,E2 300.8329} C_DIS
LIN {X -88.6423,Y 50.413,Z 106,A 146.0287,B 24.9262,C -1.9844,E1 24.8603,E2 299.4207} C_DIS
LIN {X -89.931,Y 48.0781,Z 106,A 147.5317,B 24.9265,C -1.9801,E1 24.8583,E2 297.9199} C_DIS
LIN {X -91.0786,Y 45.8669,Z 106,A 148.9412,B 24.9268,C -1.9763,E1 24.8565,E2 296.5119} C_DIS
LIN {X -92.0862,Y 43.8065,Z 106,A 150.449,B 24.9265,C -1.9801,E1 24.8547,E2 294.9869} C_DIS
LIN {X -93.7276,Y 40.1777,Z 106,A 152.6177,B 24.9272,C -1.9709,E1 24.8522,E2 292.8283} C_DIS
LIN {X -94.9297,Y 37.2433,Z 106,A 154.3819,B 24.9276,C -1.9648,E1 24.8504,E2 291.0686} C_DIS
LIN {X -96.3759,Y 33.3258,Z 106,A 156.662,B 24.9283,C -1.9552,E1 24.8483,E2 288.7985} C_DIS
LIN {X -97.2162,Y 30.7914,Z 106,A 158.1558,B 24.9287,C -1.9503,E1 24.847,E2 287.3079} C_DIS
LIN {X -98.2806,Y 27.2033,Z 106,A 160.2751,B 24.9291,C -1.9442,E1 24.8453,E2 285.1909} C_DIS
LIN {X -98.9167,Y 24.7908,Z 106,A 161.6869,B 24.9294,C -1.9401,E1 24.8444,E2 283.7806} C_DIS
LIN {X -99.4539,Y 22.535,Z 106,A 163.0111,B 24.9297,C -1.9367,E1 24.8435,E2 282.4568} C_DIS
LIN {X -100.0102,Y 19.9253,Z 106,A 164.4983,B 24.9301,C -1.9315,E1 24.8427,E2 280.9732} C_DIS
LIN {X -100.4766,Y 17.4226,Z 106,A 165.9433,B 24.9304,C -1.9274,E1 24.842,E2 279.5294} C_DIS
LIN {X -100.8732,Y 14.9562,Z 106,A 167.3592,B 24.9307,C -1.9233,E1 24.8414,E2 278.1148} C_DIS
LIN {X -101.1868,Y 12.6549,Z 106,A 168.6878,B 24.9309,C -1.9199,E1 24.8409,E2 276.7863} C_DIS
LIN {X -101.4664,Y 10.1723,Z 106,A 170.0711,B 24.9313,C -1.9147,E1 24.8405,E2 275.4072} C_DIS
LIN {X -101.6993,Y 7.5063,Z 106,A 171.6049,B 24.9315,C -1.9109,E1 24.8401,E2 273.8734} C_DIS
LIN {X -101.844,Y 5.1703,Z 106,A 172.9426,B 24.9318,C -1.9074,E1 24.8399,E2 272.5359} C_DIS
LIN {X -101.94,Y 2.674,Z 106,A 174.3328,B 24.9322,C -1.9024,E1 24.8399,E2 271.1492} C_DIS
LIN {X -101.9758,Y 0.0004,Z 106,A 175.8376,B 24.9325,C -1.8977,E1 24.8398,E2 269.6467} C_DIS
LIN {X -101.9454,Y -2.4977,Z 106,A 177.2693,B 24.9327,C -1.8941,E1 24.8398,E2 268.2148} C_DIS
LIN {X -101.8205,Y -5.5947,Z 106,A 179.1194,B 24.9329,C -1.8923,E1 24.8401,E2 266.358} C_DIS
LIN {X -101.6137,Y -8.5772,Z 106,A -179.2738,B 24.9334,C -1.8844,E1 24.8404,E2 264.7604} C_DIS
LIN {X -101.3548,Y -11.2386,Z 106,A -177.7723,B 24.9338,C -1.8795,E1 24.8409,E2 263.2614} C_DIS
LIN {X -101.0491,Y -13.7181,Z 106,A -176.3596,B 24.9341,C -1.8754,E1 24.8414,E2 261.8501} C_DIS
LIN {X -100.4739,Y -17.4384,Z 106,A -174.2313,B 24.9345,C -1.8692,E1 24.8423,E2 259.724} C_DIS
LIN {X -100.0126,Y -19.9138,Z 106,A -172.8146,B 24.9348,C -1.8648,E1 24.8431,E2 258.3093} C_DIS
LIN {X -99.5376,Y -22.1623,Z 106,A -171.4937,B 24.935,C -1.8619,E1 24.8439,E2 256.9877} C_DIS
LIN {X -98.9715,Y -24.5666,Z 106,A -170.1184,B 24.9353,C -1.8572,E1 24.8448,E2 255.6156} C_DIS
LIN {X -98.282,Y -27.1983,Z 106,A -168.5684,B 24.9356,C -1.8532,E1 24.8459,E2 254.066} C_DIS
LIN {X -97.2703,Y -30.617,Z 106,A -166.5523,B 24.936,C -1.8476,E1 24.8475,E2 252.0516} C_DIS
LIN {X -96.4928,Y -32.9854,Z 106,A -165.1296,B 24.9362,C -1.8442,E1 24.8488,E2 250.6289} C_DIS
LIN {X -95.6454,Y -35.3678,Z 106,A -163.7122,B 24.9365,C -1.8399,E1 24.8501,E2 249.2138} C_DIS
LIN {X -94.6861,Y -37.8636,Z 106,A -162.2002,B 24.9368,C -1.8358,E1 24.8517,E2 247.703} C_DIS
LIN {X -93.7301,Y -40.1716,Z 106,A -160.7884,B 24.9371,C -1.8321,E1 24.8532,E2 246.2924} C_DIS
LIN {X -92.1848,Y -43.6011,Z 106,A -158.6585,B 24.9375,C -1.8266,E1 24.8557,E2 244.1638} C_DIS
LIN {X -91.1611,Y -45.7009,Z 106,A -157.3408,B 24.9377,C -1.8232,E1 24.8573,E2 242.8473} C_DIS
LIN {X -90.1473,Y -47.6677,Z 106,A -156.0479,B 24.9378,C -1.8215,E1 24.859,E2 241.5514} C_DIS
LIN {X -88.823,Y -50.0937,Z 106,A -154.5133,B 24.9381,C -1.8166,E1 24.8611,E2 240.0204} C_DIS
LIN {X -87.4686,Y -52.4247,Z 106,A -153.0036,B 24.9384,C -1.8124,E1 24.8632,E2 238.5129} C_DIS
LIN {X -86.1582,Y -54.5514,Z 106,A -151.5922,B 24.9387,C -1.809,E1 24.8653,E2 237.1025} C_DIS
LIN {X -84.4086,Y -57.218,Z 106,A -149.7192,B 24.9387,C -1.8073,E1 24.8682,E2 235.2241} C_DIS
LIN {X -82.6395,Y -59.7479,Z 106,A -148.0473,B 24.9392,C -1.8007,E1 24.8709,E2 233.5598} C_DIS
LIN {X -80.8246,Y -62.1779,Z 106,A -146.288,B 24.9394,C -1.7985,E1 24.8739,E2 231.7972} C_DIS
LIN {X -78.7723,Y -64.7606,Z 106,A -144.2891,B 24.9394,C -1.7993,E1 24.8774,E2 229.7871} C_DIS
LIN {X -76.7511,Y -67.1416,Z 106,A -142.6161,B 24.9398,C -1.7924,E1 24.8804,E2 228.1231} C_DIS
LIN {X -73.9149,Y -70.2538,Z 106,A -140.1287,B 24.9398,C -1.7915,E1 24.8852,E2 225.6269} C_DIS
LIN {X -71.6057,Y -72.604,Z 106,A -138.3502,B 24.9403,C -1.785,E1 24.8887,E2 223.8563} C_DIS
LIN {X -68.9423,Y -75.1376,Z 106,A -136.3729,B 24.9408,C -1.7776,E1 24.8927,E2 221.8886} C_DIS
LIN {X -66.6108,Y -77.2147,Z 106,A -134.4384,B 24.9406,C -1.7806,E1 24.8968,E2 219.9392} C_DIS
LIN {X -64.2133,Y -79.2172,Z 106,A -132.7705,B 24.941,C -1.7742,E1 24.9004,E2 218.2803} C_DIS
LIN {X -61.7066,Y -81.1871,Z 106,A -130.879,B 24.941,C -1.7746,E1 24.9046,E2 216.3809} C_DIS
LIN {X -58.8549,Y -83.2768,Z 106,A -129.064,B 24.9416,C -1.765,E1 24.9086,E2 214.5825} C_DIS
LIN {X -56.798,Y -84.693,Z 106,A -127.658,B 24.9418,C -1.7628,E1 24.9119,E2 213.177} C_DIS
LIN {X -54.7069,Y -86.0585,Z 106,A -126.261,B 24.9419,C -1.7604,E1 24.9152,E2 211.7812} C_DIS
LIN {X -52.583,Y -87.3724,Z 106,A -124.8696,B 24.9421,C -1.7579,E1 24.9185,E2 210.3915} C_DIS
LIN {X -50.4247,Y -88.6355,Z 106,A -123.4326,B 24.9421,C -1.7571,E1 24.922,E2 208.9522} C_DIS
LIN {X -48.1011,Y -89.9186,Z 106,A -121.9613,B 24.9423,C -1.7543,E1 24.9256,E2 207.4832} C_DIS
LIN {X -44.8555,Y -91.5802,Z 106,A -119.8954,B 24.9424,C -1.7524,E1 24.9307,E2 205.4163} C_DIS
LIN {X -42.6225,Y -92.6404,Z 106,A -118.5012,B 24.9425,C -1.751,E1 24.9343,E2 204.022} C_DIS
LIN {X -40.1803,Y -93.7264,Z 106,A -116.996,B 24.9426,C -1.7495,E1 24.9381,E2 202.5168} C_DIS
LIN {X -37.8733,Y -94.6821,Z 106,A -115.5903,B 24.9427,C -1.7482,E1 24.9417,E2 201.1111} C_DIS
LIN {X -35.5438,Y -95.581,Z 106,A -114.1839,B 24.9428,C -1.747,E1 24.9454,E2 199.7045} C_DIS
LIN {X -33.3592,Y -96.3642,Z 106,A -112.8637,B 24.9428,C -1.7465,E1 24.9489,E2 198.383} C_DIS
LIN {X -29.618,Y -97.58,Z 106,A -110.665,B 24.943,C -1.7444,E1 24.9547,E2 196.1854} C_DIS
LIN {X -27.2319,Y -98.2725,Z 106,A -109.2773,B 24.943,C -1.7432,E1 24.9585,E2 194.7984} C_DIS
LIN {X -23.5676,Y -99.2153,Z 106,A -107.1373,B 24.943,C -1.7425,E1 24.9643,E2 192.6569} C_DIS
LIN {X -21.1303,Y -99.7627,Z 106,A -105.732,B 24.9431,C -1.7419,E1 24.9681,E2 191.2512} C_DIS
LIN {X -17.4324,Y -100.4749,Z 106,A -103.6151,B 24.9431,C -1.7412,E1 24.9739,E2 189.1339} C_DIS
LIN {X -14.966,Y -100.8718,Z 106,A -102.21,B 24.9432,C -1.7409,E1 24.9778,E2 187.7283} C_DIS
LIN {X -12.6649,Y -101.1855,Z 106,A -100.893,B 24.9432,C -1.7411,E1 24.9814,E2 186.4097} C_DIS
LIN {X -10.1828,Y -101.4653,Z 106,A -99.5001,B 24.9432,C -1.7405,E1 24.9853,E2 185.0173} C_DIS
LIN {X -7.5097,Y -101.6991,Z 106,A -97.9906,B 24.9432,C -1.7405,E1 24.9895,E2 183.5071} C_DIS
LIN {X -5.1783,Y -101.8435,Z 106,A -96.6917,B 24.9432,C -1.7401,E1 24.9931,E2 182.2088} C_DIS
LIN {X -2.685,Y -101.9397,Z 106,A -95.2923,B 24.9432,C -1.7402,E1 24.997,E2 180.8091} C_DIS
LIN {X -0.015,Y -101.9759,Z 106,A -93.7808,B 24.9432,C -1.7409,E1 25.0013,E2 179.2958} C_DIS
LIN {X -0.015,Y -101.9759,Z 106,A -93.7808,B 24.9432,C -1.7409,E1 25.0013,E2 179.2958} C_DIS
Enddeposition()
LIN {X 0.7544,Y -108.6063,Z 107,A -93.5016,B 24.9504,C -1.6274,E1 25.0013,E2 179.2859} C_DIS
Startdeposition()
$VEL.CP = VEL_PRINT
LIN {X -2.4085,Y -108.5829,Z 107,A -95.4675,B 24.9511,C -1.6148,E1 24.9957,E2 181.2816} C_DIS
LIN {X -5.0726,Y -108.4911,Z 107,A -96.8535,B 24.9511,C -1.6155,E1 24.9919,E2 182.6663} C_DIS
LIN {X -7.9899,Y -108.3166,Z 107,A -98.3953,B 24.9511,C -1.6155,E1 24.9876,E2 184.2087} C_DIS
LIN {X -10.6457,Y -108.0879,Z 107,A -99.8017,B 24.9511,C -1.6155,E1 24.9837,E2 185.6156} C_DIS
LIN {X -13.2951,Y -107.7941,Z 107,A -101.2083,B 24.9511,C -1.6157,E1 24.9798,E2 187.0228} C_DIS
LIN {X -15.6821,Y -107.4715,Z 107,A -102.4636,B 24.9511,C -1.6166,E1 24.9763,E2 188.2769} C_DIS
LIN {X -18.3149,Y -107.0543,Z 107,A -103.9066,B 24.9511,C -1.6156,E1 24.9723,E2 189.7237} C_DIS
LIN {X -21.1889,Y -106.524,Z 107,A -105.43,B 24.9511,C -1.6169,E1 24.9681,E2 191.2456} C_DIS
LIN {X -23.7968,Y -105.9719,Z 107,A -106.8375,B 24.951,C -1.6175,E1 24.9643,E2 192.6535} C_DIS
LIN {X -26.1407,Y -105.4169,Z 107,A -108.1098,B 24.951,C -1.6181,E1 24.9608,E2 193.926} C_DIS
LIN {X -28.4663,Y -104.8121,Z 107,A -109.4493,B 24.951,C -1.616,E1 24.9572,E2 195.2726} C_DIS
LIN {X -31.5281,Y -103.9342,Z 107,A -111.0619,B 24.9508,C -1.6199,E1 24.9529,E2 196.8787} C_DIS
LIN {X -33.8248,Y -103.2082,Z 107,A -112.3547,B 24.9508,C -1.6199,E1 24.9494,E2 198.1735} C_DIS
LIN {X -36.5884,Y -102.2625,Z 107,A -113.8785,B 24.9508,C -1.622,E1 24.9454,E2 199.6957} C_DIS
LIN {X -38.8482,Y -101.4242,Z 107,A -115.1525,B 24.9506,C -1.6231,E1 24.9421,E2 200.9697} C_DIS
LIN {X -41.3256,Y -100.4403,Z 107,A -116.582,B 24.9506,C -1.6235,E1 24.9384,E2 202.4011} C_DIS
LIN {X -44.7468,Y -98.9628,Z 107,A -118.605,B 24.9506,C -1.6235,E1 24.9332,E2 204.4292} C_DIS
LIN {X -47.4069,Y -97.7171,Z 107,A -120.0824,B 24.9503,C -1.6281,E1 24.9295,E2 205.8992} C_DIS
LIN {X -49.7907,Y -96.5243,Z 107,A -121.5163,B 24.9503,C -1.6288,E1 24.9259,E2 207.3354} C_DIS
LIN {X -52.3704,Y -95.1508,Z 107,A -123.0426,B 24.9501,C -1.6314,E1 24.9222,E2 208.8598} C_DIS
LIN {X -54.6898,Y -93.8369,Z 107,A -124.4529,B 24.9501,C -1.6333,E1 24.9188,E2 210.2698} C_DIS
LIN {X -56.7566,Y -92.5999,Z 107,A -125.7277,B 24.9499,C -1.635,E1 24.9157,E2 211.5445} C_DIS
LIN {X -59.2282,Y -91.0403,Z 107,A -127.2746,B 24.9498,C -1.6372,E1 24.9121,E2 213.0911} C_DIS
LIN {X -61.2319,Y -89.7035,Z 107,A -128.57,B 24.9498,C -1.6383,E1 24.9091,E2 214.3882} C_DIS
LIN {X -63.4149,Y -88.1737,Z 107,A -129.9814,B 24.9496,C -1.6405,E1 24.9059,E2 215.7994} C_DIS
LIN {X -65.7651,Y -86.4366,Z 107,A -131.5089,B 24.9494,C -1.6437,E1 24.9025,E2 217.3246} C_DIS
LIN {X -67.8666,Y -84.7966,Z 107,A -132.9206,B 24.9492,C -1.6461,E1 24.8994,E2 218.7359} C_DIS
LIN {X -69.9271,Y -83.1055,Z 107,A -134.3327,B 24.9491,C -1.6485,E1 24.8963,E2 220.1476} C_DIS
LIN {X -71.9456,Y -81.3644,Z 107,A -135.7452,B 24.9489,C -1.651,E1 24.8934,E2 221.5597} C_DIS
LIN {X -74.8916,Y -78.6611,Z 107,A -137.8639,B 24.9487,C -1.6549,E1 24.889,E2 223.6776} C_DIS
LIN {X -76.6167,Y -76.9801,Z 107,A -139.1604,B 24.9486,C -1.6567,E1 24.8865,E2 224.9755} C_DIS
LIN {X -79.3982,Y -74.1079,Z 107,A -141.2797,B 24.9483,C -1.6609,E1 24.8824,E2 227.094} C_DIS
LIN {X -81.193,Y -72.137,Z 107,A -142.6729,B 24.9481,C -1.6645,E1 24.8798,E2 228.4847} C_DIS
LIN {X -82.9389,Y -70.1227,Z 107,A -144.0861,B 24.9479,C -1.6675,E1 24.8772,E2 229.8972} C_DIS
LIN {X -84.6348,Y -68.0662,Z 107,A -145.4995,B 24.9477,C -1.6706,E1 24.8747,E2 231.3098} C_DIS
LIN {X -86.2797,Y -65.9686,Z 107,A -146.9134,B 24.9475,C -1.6737,E1 24.8723,E2 232.7231} C_DIS
LIN {X -87.8727,Y -63.8314,Z 107,A -148.3471,B 24.9474,C -1.6761,E1 24.8699,E2 234.1579} C_DIS
LIN {X -89.4127,Y -61.6556,Z 107,A -149.7611,B 24.9471,C -1.6794,E1 24.8677,E2 235.571} C_DIS
LIN {X -90.8989,Y -59.4428,Z 107,A -151.155,B 24.9469,C -1.6835,E1 24.8655,E2 236.9623} C_DIS
LIN {X -92.3588,Y -57.1485,Z 107,A -152.6109,B 24.9467,C -1.6864,E1 24.8634,E2 238.4185} C_DIS
LIN {X -93.7061,Y -54.911,Z 107,A -153.9839,B 24.9465,C -1.6903,E1 24.8614,E2 239.7894} C_DIS
LIN {X -95.1508,Y -52.3704,Z 107,A -155.535,B 24.9462,C -1.6941,E1 24.8593,E2 241.3395} C_DIS
LIN {X -96.2876,Y -50.2469,Z 107,A -156.7952,B 24.946,C -1.698,E1 24.8576,E2 242.5971} C_DIS
LIN {X -97.4917,Y -47.8687,Z 107,A -158.2478,B 24.9458,C -1.7002,E1 24.8558,E2 244.0524} C_DIS
LIN {X -98.6371,Y -45.4618,Z 107,A -159.6429,B 24.9455,C -1.7046,E1 24.8542,E2 245.4445} C_DIS
LIN {X -99.7231,Y -43.0274,Z 107,A -161.0454,B 24.9453,C -1.7088,E1 24.8526,E2 246.8448} C_DIS
LIN {X -100.8459,Y -40.3291,Z 107,A -162.6094,B 24.945,C -1.7124,E1 24.8509,E2 248.4089} C_DIS
LIN {X -102.262,Y -36.5899,Z 107,A -164.7326,B 24.9447,C -1.7181,E1 24.8489,E2 250.5304} C_DIS
LIN {X -103.047,Y -34.3128,Z 107,A -166.0314,B 24.9445,C -1.7209,E1 24.8477,E2 251.83} C_DIS
LIN {X -103.9342,Y -31.5281,Z 107,A -167.5633,B 24.9442,C -1.7259,E1 24.8464,E2 253.3588} C_DIS
LIN {X -104.6065,Y -29.2151,Z 107,A -168.8424,B 24.9439,C -1.7295,E1 24.8455,E2 254.6368} C_DIS
LIN {X -105.356,Y -26.3903,Z 107,A -170.3944,B 24.9437,C -1.7338,E1 24.8444,E2 256.1875} C_DIS
LIN {X -105.8959,Y -24.1255,Z 107,A -171.6405,B 24.9435,C -1.737,E1 24.8436,E2 257.4333} C_DIS
LIN {X -106.4362,Y -21.6163,Z 107,A -173.0195,B 24.9432,C -1.7403,E1 24.8428,E2 258.8126} C_DIS
LIN {X -106.9664,Y -18.8212,Z 107,A -174.5255,B 24.9429,C -1.7448,E1 24.8421,E2 260.3167} C_DIS
LIN {X -107.3961,Y -16.1905,Z 107,A -175.9416,B 24.9427,C -1.7489,E1 24.8414,E2 261.7315} C_DIS
LIN {X -107.7941,Y -13.2951,Z 107,A -177.4741,B 24.9423,C -1.7541,E1 24.8409,E2 263.2608} C_DIS
LIN {X -108.0612,Y -10.9013,Z 107,A -178.7535,B 24.9421,C -1.7578,E1 24.8405,E2 264.5388} C_DIS
LIN {X -108.3166,Y -7.9899,Z 107,A 179.6937,B 24.9418,C -1.7624,E1 24.8402,E2 266.0902} C_DIS
LIN {X -108.4801,Y -5.3293,Z 107,A 178.2778,B 24.9415,C -1.7665,E1 24.8399,E2 267.5047} C_DIS
LIN {X -108.5703,Y -2.9223,Z 107,A 176.9781,B 24.9413,C -1.7696,E1 24.8399,E2 268.805} C_DIS
LIN {X -108.6048,Y 1.0263,Z 107,A 174.8884,B 24.9409,C -1.7761,E1 24.8399,E2 270.8918} C_DIS
LIN {X -108.5373,Y 3.9977,Z 107,A 173.3214,B 24.9405,C -1.7811,E1 24.8399,E2 272.4561} C_DIS
LIN {X -108.4207,Y 6.4035,Z 107,A 172.0217,B 24.9403,C -1.7842,E1 24.8401,E2 273.7564} C_DIS
LIN {X -108.2309,Y 9.0624,Z 107,A 170.6054,B 24.9401,C -1.7884,E1 24.8404,E2 275.1712} C_DIS
LIN {X -107.7941,Y 13.2951,Z 107,A 168.3647,B 24.9396,C -1.7958,E1 24.8411,E2 277.4076} C_DIS
LIN {X -107.4715,Y 15.6821,Z 107,A 167.0851,B 24.9393,C -1.7996,E1 24.8416,E2 278.6858} C_DIS
LIN {X -107.0543,Y 18.3149,Z 107,A 165.6688,B 24.939,C -1.8037,E1 24.8422,E2 280.1007} C_DIS
LIN {X -106.5726,Y 20.9366,Z 107,A 164.2327,B 24.9388,C -1.8071,E1 24.843,E2 281.5371} C_DIS
LIN {X -106.0267,Y 23.5457,Z 107,A 162.8367,B 24.9385,C -1.812,E1 24.8438,E2 282.9296} C_DIS
LIN {X -105.4169,Y 26.1406,Z 107,A 161.4206,B 24.9382,C -1.8162,E1 24.8447,E2 284.3442} C_DIS
LIN {X -104.6766,Y 28.9679,Z 107,A 159.8681,B 24.9379,C -1.8206,E1 24.8459,E2 285.895} C_DIS
LIN {X -103.9342,Y 31.5281,Z 107,A 158.4524,B 24.9376,C -1.8247,E1 24.847,E2 287.3092} C_DIS
LIN {X -103.1291,Y 34.0693,Z 107,A 157.0366,B 24.9373,C -1.8288,E1 24.8482,E2 288.7234} C_DIS
LIN {X -102.262,Y 36.5899,Z 107,A 155.6207,B 24.937,C -1.8328,E1 24.8495,E2 290.1378} C_DIS
LIN {X -101.4242,Y 38.8482,Z 107,A 154.3415,B 24.9368,C -1.8364,E1 24.8508,E2 291.4155} C_DIS
LIN {X -100.3434,Y 41.5636,Z 107,A 152.789,B 24.9365,C -1.8408,E1 24.8524,E2 292.9664} C_DIS
LIN {X -98.7456,Y 45.2288,Z 107,A 150.6658,B 24.9361,C -1.8466,E1 24.8548,E2 295.0872} C_DIS
LIN {X -97.7171,Y 47.4069,Z 107,A 149.3868,B 24.9358,C -1.8502,E1 24.8563,E2 296.3647} C_DIS
LIN {X -96.4073,Y 50.0195,Z 107,A 147.8352,B 24.9355,C -1.8544,E1 24.8583,E2 297.9147} C_DIS
LIN {X -94.6262,Y 53.3098,Z 107,A 145.8286,B 24.9352,C -1.859,E1 24.861,E2 299.9209} C_DIS
LIN {X -93.1587,Y 55.8372,Z 107,A 144.2971,B 24.9349,C -1.8638,E1 24.8632,E2 301.4489} C_DIS
LIN {X -91.8911,Y 57.8972,Z 107,A 142.9945,B 24.9347,C -1.8664,E1 24.8651,E2 302.7517} C_DIS
LIN {X -90.3067,Y 60.341,Z 107,A 141.4673,B 24.9344,C -1.8711,E1 24.8674,E2 304.2755} C_DIS
LIN {X -88.9453,Y 62.3281,Z 107,A 140.1889,B 24.9341,C -1.8743,E1 24.8694,E2 305.5525} C_DIS
LIN {X -87.2371,Y 64.6994,Z 107,A 138.6382,B 24.9339,C -1.8782,E1 24.872,E2 307.1016} C_DIS
LIN {X -85.623,Y 66.8209,Z 107,A 137.2235,B 24.9336,C -1.8816,E1 24.8744,E2 308.5147} C_DIS
LIN {X -83.998,Y 68.8518,Z 107,A 135.8505,B 24.9334,C -1.8852,E1 24.8768,E2 309.8856} C_DIS
LIN {X -82.4078,Y 70.7461,Z 107,A 134.5313,B 24.9332,C -1.8881,E1 24.8792,E2 311.204} C_DIS
LIN {X -80.4754,Y 72.9386,Z 107,A 132.981,B 24.9329,C -1.8917,E1 24.8821,E2 312.7527} C_DIS
LIN {X -78.6611,Y 74.8916,Z 107,A 131.5671,B 24.9327,C -1.8949,E1 24.8848,E2 314.1651} C_DIS
LIN {X -76.0341,Y 77.5556,Z 107,A 129.5828,B 24.9324,C -1.8993,E1 24.8887,E2 316.1473} C_DIS
LIN {X -74.1079,Y 79.3982,Z 107,A 128.1494,B 24.9322,C -1.9016,E1 24.8916,E2 317.5811} C_DIS
LIN {X -72.137,Y 81.193,Z 107,A 126.756,B 24.9319,C -1.9053,E1 24.8945,E2 318.9712} C_DIS
LIN {X -70.1227,Y 82.9389,Z 107,A 125.343,B 24.9317,C -1.9082,E1 24.8975,E2 320.3828} C_DIS
LIN {X -68.0662,Y 84.6348,Z 107,A 123.93,B 24.9315,C -1.9111,E1 24.9005,E2 321.7943} C_DIS
LIN {X -65.9686,Y 86.2797,Z 107,A 122.5171,B 24.9313,C -1.9138,E1 24.9036,E2 323.2059} C_DIS
LIN {X -63.8314,Y 87.8727,Z 107,A 121.0846,B 24.9312,C -1.9157,E1 24.9069,E2 324.6389} C_DIS
LIN {X -61.6556,Y 89.4127,Z 107,A 119.6723,B 24.931,C -1.9183,E1 24.9101,E2 326.0499} C_DIS
LIN {X -59.4428,Y 90.8989,Z 107,A 118.2802,B 24.9308,C -1.9216,E1 24.9133,E2 327.4388} C_DIS
LIN {X -56.9762,Y 92.4665,Z 107,A 116.7321,B 24.9306,C -1.9242,E1 24.917,E2 328.9855} C_DIS
LIN {X -54.911,Y 93.7061,Z 107,A 115.436,B 24.9305,C -1.9256,E1 24.9201,E2 330.2822} C_DIS
LIN {X -52.3704,Y 95.1508,Z 107,A 113.9083,B 24.9303,C -1.9288,E1 24.9238,E2 331.8067} C_DIS
LIN {X -50.2469,Y 96.2876,Z 107,A 112.6333,B 24.9301,C -1.9308,E1 24.927,E2 333.0805} C_DIS
LIN {X -47.8687,Y 97.4917,Z 107,A 111.2021,B 24.9301,C -1.9321,E1 24.9305,E2 334.5124} C_DIS
LIN {X -45.4618,Y 98.6371,Z 107,A 109.8109,B 24.9298,C -1.9349,E1 24.9341,E2 335.9005} C_DIS
LIN {X -42.7918,Y 99.8258,Z 107,A 108.2644,B 24.9297,C -1.937,E1 24.938,E2 337.4458} C_DIS
LIN {X -40.3291,Y 100.8459,Z 107,A 106.8537,B 24.9295,C -1.9388,E1 24.9417,E2 338.8553} C_DIS
LIN {X -37.8421,Y 101.8052,Z 107,A 105.4436,B 24.9295,C -1.9405,E1 24.9453,E2 340.2643} C_DIS
LIN {X -35.5747,Y 102.6182,Z 107,A 104.1694,B 24.9293,C -1.942,E1 24.9487,E2 341.5375} C_DIS
LIN {X -33.0628,Y 103.4548,Z 107,A 102.7462,B 24.9293,C -1.9426,E1 24.9525,E2 342.9618} C_DIS
LIN {X -30.4966,Y 104.2401,Z 107,A 101.3498,B 24.9291,C -1.9449,E1 24.9562,E2 344.355} C_DIS
LIN {X -27.6812,Y 105.0242,Z 107,A 99.8047,B 24.929,C -1.9464,E1 24.9604,E2 345.899} C_DIS
LIN {X -25.0954,Y 105.6719,Z 107,A 98.3953,B 24.9289,C -1.9476,E1 24.9642,E2 347.3074} C_DIS
LIN {X -22.7456,Y 106.2012,Z 107,A 97.1022,B 24.9289,C -1.9478,E1 24.9677,E2 348.6016} C_DIS
LIN {X -20.1325,Y 106.7274,Z 107,A 95.7134,B 24.9287,C -1.9497,E1 24.9715,E2 349.9876} C_DIS
LIN {X -17.2537,Y 107.2317,Z 107,A 94.1692,B 24.9287,C -1.9507,E1 24.9758,E2 351.5308} C_DIS
LIN {X -15.0223,Y 107.5652,Z 107,A 92.9309,B 24.9287,C -1.9496,E1 24.9792,E2 352.7728} C_DIS
LIN {X -12.2266,Y 107.9192,Z 107,A 91.4888,B 24.9285,C -1.9522,E1 24.9832,E2 354.2097} C_DIS
LIN {X -9.3185,Y 108.2104,Z 107,A 89.9455,B 24.9285,C -1.9529,E1 24.9875,E2 355.7522} C_DIS
LIN {X -6.9165,Y 108.3892,Z 107,A 88.6536,B 24.9285,C -1.9526,E1 24.9911,E2 357.0452} C_DIS
LIN {X -3.9977,Y 108.5373,Z 107,A 87.1306,B 24.9285,C -1.9538,E1 24.9953,E2 358.5655} C_DIS
LIN {X -1.3328,Y 108.6027,Z 107,A 85.7234,B 24.9285,C -1.9542,E1 24.9992,E2 359.9721} C_DIS
LIN {X 1.3206,Y 108.6027,Z 107,A 84.3246,B 24.9284,C -1.9544,E1 25.0031,E2 361.3701} C_DIS
LIN {X 3.9977,Y 108.5373,Z 107,A 82.9102,B 24.9284,C -1.9545,E1 25.0071,E2 362.7841} C_DIS
LIN {X 6.4035,Y 108.4207,Z 107,A 81.6195,B 24.9284,C -1.9538,E1 25.0107,E2 364.0761} C_DIS
LIN {X 9.0624,Y 108.2309,Z 107,A 80.2133,B 24.9284,C -1.9537,E1 25.0146,E2 365.4818} C_DIS
LIN {X 11.9713,Y 107.9491,Z 107,A 78.6921,B 24.9284,C -1.9543,E1 25.0188,E2 367.0005} C_DIS
LIN {X 14.1967,Y 107.6773,Z 107,A 77.487,B 24.9284,C -1.9531,E1 25.0222,E2 368.2074} C_DIS
LIN {X 16.9998,Y 107.271,Z 107,A 76.0162,B 24.9284,C -1.9536,E1 25.0262,E2 369.6756} C_DIS
LIN {X 19.7343,Y 106.8022,Z 107,A 74.547,B 24.9284,C -1.9529,E1 25.0302,E2 371.1451} C_DIS
LIN {X 22.2428,Y 106.3076,Z 107,A 73.1867,B 24.9286,C -1.9518,E1 25.034,E2 372.5063} C_DIS
LIN {X 26.1407,Y 105.4169,Z 107,A 71.0796,B 24.9286,C -1.9507,E1 25.0397,E2 374.6129} C_DIS
LIN {X 28.9679,Y 104.6766,Z 107,A 69.5599,B 24.9286,C -1.9507,E1 25.0438,E2 376.1304} C_DIS
LIN {X 31.2817,Y 104.0072,Z 107,A 68.2913,B 24.9287,C -1.9498,E1 25.0472,E2 377.3989} C_DIS
LIN {X 33.6055,Y 103.2792,Z 107,A 66.9497,B 24.929,C -1.9464,E1 25.0508,E2 378.7459} C_DIS
LIN {X 36.5899,Y 102.262,Z 107,A 65.3484,B 24.9289,C -1.9475,E1 25.055,E2 380.3414} C_DIS
LIN {X 40.0899,Y 100.9398,Z 107,A 63.3788,B 24.929,C -1.9458,E1 25.0601,E2 382.3109} C_DIS
LIN {X 42.7918,Y 99.8258,Z 107,A 61.8407,B 24.9291,C -1.9442,E1 25.0641,E2 383.8489} C_DIS
LIN {X 44.9945,Y 98.8511,Z 107,A 60.5731,B 24.9292,C -1.9429,E1 25.0673,E2 385.1166} C_DIS
LIN {X 47.4069,Y 97.7171,Z 107,A 59.1508,B 24.9294,C -1.9406,E1 25.0709,E2 386.5407} C_DIS
LIN {X 49.7199,Y 96.5604,Z 107,A 57.801,B 24.9294,C -1.9394,E1 25.0743,E2 387.8896} C_DIS
LIN {X 52.1445,Y 95.2733,Z 107,A 56.3462,B 24.9296,C -1.9372,E1 25.0778,E2 389.3455} C_DIS
LIN {X 54.6898,Y 93.8369,Z 107,A 54.8291,B 24.9297,C -1.9359,E1 25.0815,E2 390.861} C_DIS
LIN {X 56.9762,Y 92.4665,Z 107,A 53.4275,B 24.9299,C -1.934,E1 25.0848,E2 392.2627} C_DIS
LIN {X 59.012,Y 91.1791,Z 107,A 52.1412,B 24.9301,C -1.9314,E1 25.0879,E2 393.5511} C_DIS
LIN {X 61.4446,Y 89.5594,Z 107,A 50.625,B 24.9301,C -1.9299,E1 25.0914,E2 395.0657} C_DIS
LIN {X 63.4149,Y 88.1737,Z 107,A 49.3389,B 24.9304,C -1.9271,E1 25.0943,E2 396.354} C_DIS
LIN {X 65.5596,Y 86.5909,Z 107,A 47.958,B 24.9304,C -1.9257,E1 25.0974,E2 397.7333} C_DIS
LIN {X 67.665,Y 84.9559,Z 107,A 46.5374,B 24.9307,C -1.9225,E1 25.1005,E2 399.1562} C_DIS
LIN {X 69.7295,Y 83.2697,Z 107,A 45.137,B 24.9309,C -1.92,E1 25.1035,E2 400.557} C_DIS
LIN {X 71.752,Y 81.5334,Z 107,A 43.7567,B 24.931,C -1.9184,E1 25.1064,E2 401.9358} C_DIS
LIN {X 73.7314,Y 79.748,Z 107,A 42.3563,B 24.9312,C -1.9157,E1 25.1093,E2 403.3367} C_DIS
LIN {X 75.6663,Y 77.9145,Z 107,A 40.9367,B 24.9314,C -1.9122,E1 25.1122,E2 404.7587} C_DIS
LIN {X 77.7362,Y 75.8513,Z 107,A 39.4219,B 24.9316,C -1.91,E1 25.1152,E2 406.2723} C_DIS
LIN {X 79.3982,Y 74.1079,Z 107,A 38.1741,B 24.9317,C -1.9082,E1 25.1176,E2 407.5189} C_DIS
LIN {X 81.193,Y 72.137,Z 107,A 36.7722,B 24.932,C -1.9052,E1 25.1202,E2 408.9217} C_DIS
LIN {X 83.1055,Y 69.9271,Z 107,A 35.2236,B 24.9322,C -1.9013,E1 25.123,E2 410.4724} C_DIS
LIN {X 84.7966,Y 67.8666,Z 107,A 33.8248,B 24.9324,C -1.8983,E1 25.1255,E2 411.8719} C_DIS
LIN {X 86.2797,Y 65.9686,Z 107,A 32.5607,B 24.9326,C -1.8955,E1 25.1276,E2 413.1367} C_DIS
LIN {X 87.8727,Y 63.8314,Z 107,A 31.1423,B 24.9329,C -1.8915,E1 25.13,E2 414.5577} C_DIS
LIN {X 89.5594,Y 61.4446,Z 107,A 29.6289,B 24.9331,C -1.8887,E1 25.1324,E2 416.0701} C_DIS
LIN {X 91.0403,Y 59.2282,Z 107,A 28.2302,B 24.9334,C -1.8854,E1 25.1345,E2 417.4697} C_DIS
LIN {X 92.3303,Y 57.1941,Z 107,A 26.9863,B 24.9335,C -1.8832,E1 25.1364,E2 418.7124} C_DIS
LIN {X 93.7061,Y 54.911,Z 107,A 25.5687,B 24.9338,C -1.879,E1 25.1384,E2 420.1328} C_DIS
LIN {X 95.2733,Y 52.1445,Z 107,A 23.7879,B 24.9345,C -1.8699,E1 25.1409,E2 421.9256} C_DIS
LIN {X 96.8369,Y 49.179,Z 107,A 22.1011,B 24.9345,C -1.8686,E1 25.143,E2 423.6067} C_DIS
LIN {X 98.0718,Y 46.6688,Z 107,A 20.6563,B 24.9347,C -1.8657,E1 25.1448,E2 425.0505} C_DIS
LIN {X 99.1876,Y 44.2479,Z 107,A 19.2785,B 24.9349,C -1.8629,E1 25.1464,E2 426.4274} C_DIS
LIN {X 100.3434,Y 41.5636,Z 107,A 17.7463,B 24.9352,C -1.8589,E1 25.148,E2 427.9609} C_DIS
LIN {X 101.3332,Y 39.0885,Z 107,A 16.349,B 24.9355,C -1.8551,E1 25.1495,E2 429.3592} C_DIS
LIN {X 102.6182,Y 35.5747,Z 107,A 14.388,B 24.9359,C -1.8498,E1 25.1513,E2 431.3217} C_DIS
LIN {X 103.5394,Y 32.8011,Z 107,A 12.8559,B 24.9362,C -1.8456,E1 25.1526,E2 432.8552} C_DIS
LIN {X 104.2401,Y 30.4966,Z 107,A 11.5937,B 24.9364,C -1.8421,E1 25.1536,E2 434.1184} C_DIS
LIN {X 104.9572,Y 27.9293,Z 107,A 10.1768,B 24.9367,C -1.8373,E1 25.1547,E2 435.5384} C_DIS
LIN {X 105.611,Y 25.3451,Z 107,A 8.8134,B 24.9369,C -1.8348,E1 25.1556,E2 436.8998} C_DIS
LIN {X 106.2012,Y 22.7456,Z 107,A 7.4029,B 24.9372,C -1.8303,E1 25.1564,E2 438.3128} C_DIS
LIN {X 106.7274,Y 20.1325,Z 107,A 6.0064,B 24.9375,C -1.8263,E1 25.1572,E2 439.7106} C_DIS
LIN {X 107.2317,Y 17.2537,Z 107,A 4.4748,B 24.9378,C -1.8218,E1 25.1579,E2 441.2437} C_DIS
LIN {X 107.7279,Y 13.8062,Z 107,A 2.6097,B 24.9383,C -1.8148,E1 25.1586,E2 443.1143} C_DIS
LIN {X 108.0612,Y 10.9013,Z 107,A 1.1179,B 24.9385,C -1.8121,E1 25.1591,E2 444.6038} C_DIS
LIN {X 108.3166,Y 7.9899,Z 107,A -0.4135,B 24.9388,C -1.8076,E1 25.1594,E2 446.1367} C_DIS
LIN {X 108.4801,Y 5.3293,Z 107,A -1.8099,B 24.939,C -1.8035,E1 25.1596,E2 447.5345} C_DIS
LIN {X 108.5703,Y 2.9223,Z 107,A -3.0915,B 24.9393,C -1.7989,E1 25.1598,E2 448.8192} C_DIS
LIN {X 108.6104,Y 0,Z 107,A -4.5675,B 24.9395,C -1.7968,E1 25.1598,E2 450.2914} C_DIS
LIN {X 108.5829,Y -2.4085,Z 107,A -5.8845,B 24.9399,C -1.7907,E1 25.1598,E2 451.615} C_DIS
LIN {X 108.4911,Y -5.0726,Z 107,A -7.2611,B 24.9401,C -1.7874,E1 25.1596,E2 452.9912} C_DIS
LIN {X 108.3587,Y -7.3679,Z 107,A -8.5298,B 24.9405,C -1.781,E1 25.1593,E2 454.2673} C_DIS
LIN {X 108.0879,Y -10.6457,Z 107,A -10.1884,B 24.9407,C -1.7787,E1 25.1589,E2 455.9216} C_DIS
LIN {X 107.7941,Y -13.2951,Z 107,A -11.585,B 24.941,C -1.7746,E1 25.1585,E2 457.3197} C_DIS
LIN {X 107.4715,Y -15.6821,Z 107,A -12.8666,B 24.9413,C -1.77,E1 25.158,E2 458.6045} C_DIS
LIN {X 107.0543,Y -18.3149,Z 107,A -14.263,B 24.9416,C -1.7659,E1 25.1573,E2 460.0024} C_DIS
LIN {X 106.3076,Y -22.2428,Z 107,A -16.3578,B 24.942,C -1.7597,E1 25.1562,E2 462.0995} C_DIS
LIN {X 105.7297,Y -24.8451,Z 107,A -17.7345,B 24.9422,C -1.7565,E1 25.1554,E2 463.4758} C_DIS
LIN {X 105.0882,Y -27.4323,Z 107,A -19.1511,B 24.9425,C -1.7516,E1 25.1544,E2 464.8959} C_DIS
LIN {X 104.3132,Y -30.2503,Z 107,A -20.6623,B 24.9427,C -1.748,E1 25.1532,E2 466.4069} C_DIS
LIN {X 103.6155,Y -32.5557,Z 107,A -21.9246,B 24.943,C -1.7444,E1 25.1522,E2 467.6705} C_DIS
LIN {X 102.7033,Y -35.3322,Z 107,A -23.4559,B 24.9433,C -1.74,E1 25.1508,E2 469.2036} C_DIS
LIN {X 101.4242,Y -38.8482,Z 107,A -25.4165,B 24.9436,C -1.7344,E1 25.1489,E2 471.1663} C_DIS
LIN {X 100.4403,Y -41.3256,Z 107,A -26.8283,B 24.9439,C -1.7298,E1 25.1474,E2 472.5811} C_DIS
LIN {X 99.2931,Y -44.0136,Z 107,A -28.3448,B 24.9442,C -1.7262,E1 25.1458,E2 474.0979} C_DIS
LIN {X 98.1831,Y -46.4371,Z 107,A -29.7424,B 24.9444,C -1.7223,E1 25.1441,E2 475.4971} C_DIS
LIN {X 97.1485,Y -48.5612,Z 107,A -30.9854,B 24.9446,C -1.7187,E1 25.1426,E2 476.7419} C_DIS
LIN {X 95.7863,Y -51.1988,Z 107,A -32.5364,B 24.9449,C -1.7147,E1 25.1406,E2 478.2942} C_DIS
LIN {X 94.6262,Y -53.3098,Z 107,A -33.8192,B 24.9452,C -1.7105,E1 25.1388,E2 479.5803} C_DIS
LIN {X 93.1587,Y -55.8372,Z 107,A -35.3317,B 24.9454,C -1.7072,E1 25.1367,E2 481.0927} C_DIS
LIN {X 91.8965,Y -57.8886,Z 107,A -36.6143,B 24.9456,C -1.7031,E1 25.1348,E2 482.3786} C_DIS
LIN {X 89.7035,Y -61.2319,Z 107,A -38.7044,B 24.946,C -1.698,E1 25.1315,E2 484.4703} C_DIS
LIN {X 88.1737,Y -63.4149,Z 107,A -40.1087,B 24.9462,C -1.6941,E1 25.1293,E2 485.8768} C_DIS
LIN {X 86.4366,Y -65.7651,Z 107,A -41.6215,B 24.9464,C -1.6912,E1 25.1267,E2 487.3893} C_DIS
LIN {X 84.7966,Y -67.8666,Z 107,A -43.0195,B 24.9466,C -1.6878,E1 25.1243,E2 488.7889} C_DIS
LIN {X 83.152,Y -69.8712,Z 107,A -44.3816,B 24.9468,C -1.6844,E1 25.1219,E2 490.1526} C_DIS
LIN {X 81.3644,Y -71.9456,Z 107,A -45.8162,B 24.947,C -1.6811,E1 25.1192,E2 491.5886} C_DIS
LIN {X 78.703,Y -74.8471,Z 107,A -47.8836,B 24.9473,C -1.6763,E1 25.1153,E2 493.6583} C_DIS
LIN {X 76.9801,Y -76.6167,Z 107,A -49.1981,B 24.9476,C -1.6726,E1 25.1127,E2 494.9759} C_DIS
LIN {X 74.1079,Y -79.3982,Z 107,A -51.2965,B 24.9479,C -1.668,E1 25.1085,E2 497.0765} C_DIS
LIN {X 72.137,Y -81.193,Z 107,A -52.676,B 24.9479,C -1.6658,E1 25.1056,E2 498.4555} C_DIS
LIN {X 70.1227,Y -82.9389,Z 107,A -54.0752,B 24.9482,C -1.6629,E1 25.1027,E2 499.8562} C_DIS
LIN {X 68.0662,Y -84.6348,Z 107,A -55.4746,B 24.9484,C -1.6601,E1 25.0996,E2 501.2569} C_DIS
LIN {X 65.9686,Y -86.2797,Z 107,A -56.8746,B 24.9485,C -1.6573,E1 25.0965,E2 502.6583} C_DIS
LIN {X 63.8314,Y -87.8727,Z 107,A -58.2941,B 24.9487,C -1.6538,E1 25.0933,E2 504.0811} C_DIS
LIN {X 61.6556,Y -89.4127,Z 107,A -59.6942,B 24.9489,C -1.6512,E1 25.0901,E2 505.4825} C_DIS
LIN {X 59.4428,Y -90.8989,Z 107,A -61.0745,B 24.949,C -1.6495,E1 25.0869,E2 506.8622} C_DIS
LIN {X 57.1104,Y -92.3826,Z 107,A -62.5347,B 24.9492,C -1.6466,E1 25.0835,E2 508.3246} C_DIS
LIN {X 54.911,Y -93.7061,Z 107,A -63.8757,B 24.9493,C -1.6447,E1 25.0802,E2 509.6661} C_DIS
LIN {X 52.3704,Y -95.1508,Z 107,A -65.4118,B 24.9495,C -1.6421,E1 25.0765,E2 511.2036} C_DIS
LIN {X 50.2469,Y -96.2876,Z 107,A -66.6974,B 24.9496,C -1.6393,E1 25.0733,E2 512.4922} C_DIS
LIN {X 47.8687,Y -97.4917,Z 107,A -68.0985,B 24.9498,C -1.6372,E1 25.0698,E2 513.8946} C_DIS
LIN {X 45.4618,Y -98.6371,Z 107,A -69.4803,B 24.9498,C -1.636,E1 25.0663,E2 515.2756} C_DIS
LIN {X 43.0274,Y -99.7231,Z 107,A -70.8819,B 24.95,C -1.6341,E1 25.0627,E2 516.6784} C_DIS
LIN {X 40.3291,Y -100.8459,Z 107,A -72.4189,B 24.95,C -1.6321,E1 25.0587,E2 518.2167} C_DIS
LIN {X 37.8421,Y -101.8052,Z 107,A -73.8208,B 24.9502,C -1.6303,E1 25.0551,E2 519.6197} C_DIS
LIN {X 35.5747,Y -102.6182,Z 107,A -75.0881,B 24.9502,C -1.6288,E1 25.0517,E2 520.8878} C_DIS
LIN {X 32.8011,Y -103.5394,Z 107,A -76.7874,B 24.9508,C -1.6203,E1 25.0472,E2 522.6041} C_DIS
LIN {X 29.5238,Y -104.5191,Z 107,A -78.4799,B 24.9506,C -1.623,E1 25.0427,E2 524.2873} C_DIS
LIN {X 26.3903,Y -105.356,Z 107,A -80.1332,B 24.9506,C -1.6236,E1 25.0382,E2 525.9367} C_DIS
LIN {X 23.7968,Y -105.9719,Z 107,A -81.5368,B 24.9506,C -1.6224,E1 25.0344,E2 527.3413} C_DIS
LIN {X 21.1889,Y -106.524,Z 107,A -82.9403,B 24.9507,C -1.6213,E1 25.0306,E2 528.7457} C_DIS
LIN {X 18.8212,Y -106.9664,Z 107,A -84.2284,B 24.9509,C -1.6195,E1 25.027,E2 530.0365} C_DIS
LIN {X 16.3356,Y -107.3737,Z 107,A -85.5804,B 24.9509,C -1.6176,E1 25.0233,E2 531.3918} C_DIS
LIN {X 13.2951,Y -107.7941,Z 107,A -87.1525,B 24.9509,C -1.6185,E1 25.0189,E2 532.9605} C_DIS
LIN {X 10.9013,Y -108.0612,Z 107,A -88.4215,B 24.9509,C -1.6178,E1 25.0154,E2 534.2301} C_DIS
LIN {X 7.9899,Y -108.3166,Z 107,A -89.9618,B 24.951,C -1.6171,E1 25.0111,E2 535.7714} C_DIS
LIN {X 5.3293,Y -108.4801,Z 107,A -91.3666,B 24.951,C -1.6166,E1 25.0072,E2 537.1769} C_DIS
LIN {X 3.1516,Y -108.5633,Z 107,A -92.578,B 24.9512,C -1.6137,E1 25.0038,E2 538.3949} C_DIS
LIN {X 0.7544,Y -108.6063,Z 107,A -93.5016,B 24.9504,C -1.6274,E1 25.0013,E2 539.2859} C_DIS
Enddeposition()
LIN {X 0.7544,Y -108.6063,Z 107,A -93.5016,B 24.9504,C -1.6274,E1 25.0013,E2 539.2859} C_DIS
Startdeposition()
$VEL.CP = VEL_PRINT
LIN {X 1.3485,Y -107.6372,Z 107,A -92.7093,B 24.9481,C -1.6638,E1 25.0038,E2 538.4073} C_DIS
LIN {X 4.706,Y -107.5409,Z 107,A -91.0207,B 24.9483,C -1.6604,E1 25.0084,E2 536.7272} C_DIS
LIN {X 9.3773,Y -107.2358,Z 107,A -88.3953,B 24.9479,C -1.6671,E1 25.0158,E2 534.0872} C_DIS
LIN {X 14.0002,Y -106.7296,Z 107,A -85.7723,B 24.9474,C -1.6748,E1 25.0231,E2 531.4481} C_DIS
LIN {X 17.6955,Y -106.1794,Z 107,A -83.4136,B 24.9464,C -1.6918,E1 25.0297,E2 529.0513} C_DIS
LIN {X 21.8835,Y -105.3962,Z 107,A -81.6733,B 24.9476,C -1.6716,E1 25.0343,E2 527.3611} C_DIS
LIN {X 25.2153,Y -104.6493,Z 107,A -80.1216,B 24.9482,C -1.6622,E1 25.0385,E2 525.8338} C_DIS
LIN {X 27.8738,Y -103.9725,Z 107,A -78.5297,B 24.9478,C -1.6692,E1 25.0428,E2 524.2277} C_DIS
LIN {X 30.4031,Y -103.2613,Z 107,A -76.9608,B 24.9472,C -1.678,E1 25.0471,E2 522.6408} C_DIS
LIN {X 33.9845,Y -102.1393,Z 107,A -75.2468,B 24.9478,C -1.6684,E1 25.0516,E2 520.9526} C_DIS
LIN {X 36.843,Y -101.1424,Z 107,A -73.5033,B 24.9474,C -1.6761,E1 25.0562,E2 519.1944} C_DIS
LIN {X 40.3686,Y -99.7879,Z 107,A -71.5679,B 24.9474,C -1.6758,E1 25.0612,E2 517.2642} C_DIS
LIN {X 43.3412,Y -98.5335,Z 107,A -69.5952,B 24.9465,C -1.6892,E1 25.0663,E2 515.2645} C_DIS
LIN {X 47.4581,Y -96.6182,Z 107,A -67.5992,B 24.9474,C -1.6751,E1 25.0713,E2 513.3069} C_DIS
LIN {X 51.7767,Y -94.375,Z 107,A -64.876,B 24.9468,C -1.6852,E1 25.0781,E2 510.5676} C_DIS
LIN {X 54.6886,Y -92.7165,Z 107,A -63.1011,B 24.9466,C -1.6881,E1 25.0823,E2 508.7912} C_DIS
LIN {X 57.2069,Y -91.1845,Z 107,A -61.1453,B 24.9453,C -1.7077,E1 25.0871,E2 506.7953} C_DIS
LIN {X 60.9039,Y -88.7592,Z 107,A -59.0126,B 24.9457,C -1.7028,E1 25.092,E2 504.6812} C_DIS
LIN {X 64.037,Y -86.5261,Z 107,A -57.0061,B 24.9455,C -1.7053,E1 25.0965,E2 502.6759} C_DIS
LIN {X 66.8219,Y -84.3922,Z 107,A -55.1595,B 24.9453,C -1.7085,E1 25.1006,E2 500.8286} C_DIS
LIN {X 70.3071,Y -81.514,Z 107,A -52.7845,B 24.945,C -1.7126,E1 25.1056,E2 498.4532} C_DIS
LIN {X 72.297,Y -79.7543,Z 107,A -51.2967,B 24.9446,C -1.7191,E1 25.1087,E2 496.956} C_DIS
LIN {X 75.0274,Y -77.1899,Z 107,A -49.347,B 24.9444,C -1.722,E1 25.1127,E2 495.0076} C_DIS
LIN {X 77.1549,Y -75.0637,Z 107,A -47.7011,B 24.944,C -1.7279,E1 25.1159,E2 493.3547} C_DIS
LIN {X 80.148,Y -71.8574,Z 107,A -45.5346,B 24.9441,C -1.7265,E1 25.12,E2 491.201} C_DIS
LIN {X 82.4447,Y -69.2124,Z 107,A -43.6126,B 24.9437,C -1.7339,E1 25.1235,E2 489.2704} C_DIS
LIN {X 85.3113,Y -65.6444,Z 107,A -40.1715,B 24.9403,C -1.7848,E1 25.1295,E2 485.7253} C_DIS
LIN {X 88.9235,Y -60.6625,Z 107,A -38.2119,B 24.9435,C -1.7358,E1 25.1325,E2 483.8909} C_DIS
LIN {X 91.9283,Y -56.0035,Z 107,A -35.0015,B 24.9422,C -1.7556,E1 25.1373,E2 480.6501} C_DIS
LIN {X 93.8837,Y -52.6602,Z 107,A -33.0599,B 24.9422,C -1.7563,E1 25.14,E2 478.7168} C_DIS
LIN {X 95.0298,Y -50.5642,Z 107,A -31.6389,B 24.9415,C -1.7666,E1 25.1419,E2 477.2789} C_DIS
LIN {X 96.8753,Y -46.9307,Z 107,A -29.7312,B 24.9418,C -1.7616,E1 25.1442,E2 475.3932} C_DIS
LIN {X 98.1217,Y -44.2642,Z 107,A -28.0352,B 24.9411,C -1.7721,E1 25.1462,E2 473.6817} C_DIS
LIN {X 99.3464,Y -41.4444,Z 107,A -26.3338,B 24.9406,C -1.78,E1 25.1481,E2 471.971} C_DIS
LIN {X 100.4414,Y -38.7182,Z 107,A -24.8219,B 24.9404,C -1.7825,E1 25.1496,E2 470.4615} C_DIS
LIN {X 101.6842,Y -35.3219,Z 107,A -22.8381,B 24.9399,C -1.7911,E1 25.1515,E2 468.4685} C_DIS
LIN {X 102.8379,Y -31.8051,Z 107,A -20.9866,B 24.9399,C -1.7921,E1 25.1531,E2 466.6252} C_DIS
LIN {X 103.7343,Y -28.7535,Z 107,A -19.3905,B 24.9397,C -1.7932,E1 25.1543,E2 465.0357} C_DIS
LIN {X 105.2584,Y -22.5397,Z 107,A -15.8332,B 24.9385,C -1.8108,E1 25.1566,E2 461.4576} C_DIS
LIN {X 106.0359,Y -18.5427,Z 107,A -13.6901,B 24.9381,C -1.8167,E1 25.1577,E2 459.3131} C_DIS
LIN {X 106.5152,Y -15.5527,Z 107,A -12.107,B 24.9379,C -1.8206,E1 25.1583,E2 457.73} C_DIS
LIN {X 106.9548,Y -12.1651,Z 107,A -10.382,B 24.9377,C -1.8224,E1 25.1589,E2 456.011} C_DIS
LIN {X 107.3417,Y -8.075,Z 107,A -8.2434,B 24.9374,C -1.8274,E1 25.1594,E2 453.8734} C_DIS
LIN {X 107.5271,Y -5.0287,Z 107,A -6.4918,B 24.9367,C -1.8383,E1 25.1597,E2 452.1065} C_DIS
LIN {X 107.6323,Y -1.6169,Z 107,A -4.7405,B 24.9365,C -1.8413,E1 25.1597,E2 450.3586} C_DIS
LIN {X 107.6254,Y 1.9917,Z 107,A -2.8299,B 24.9361,C -1.847,E1 25.1597,E2 448.4457} C_DIS
LIN {X 107.483,Y 5.8814,Z 107,A -0.8195,B 24.9358,C -1.851,E1 25.1595,E2 446.4378} C_DIS
LIN {X 107.1177,Y 10.6446,Z 107,A 1.846,B 24.9348,C -1.8646,E1 25.1588,E2 443.7563} C_DIS
LIN {X 106.662,Y 14.5194,Z 107,A 4.2336,B 24.9334,C -1.8849,E1 25.158,E2 441.3348} C_DIS
LIN {X 106.1406,Y 17.9276,Z 107,A 6.16,B 24.9327,C -1.8948,E1 25.157,E2 439.3963} C_DIS
LIN {X 105.4042,Y 21.8445,Z 107,A 7.9654,B 24.9332,C -1.8874,E1 25.156,E2 437.6189} C_DIS
LIN {X 104.0363,Y 27.6379,Z 107,A 10.8772,B 24.9333,C -1.8859,E1 25.1541,E2 434.7275} C_DIS
LIN {X 103.2756,Y 30.3547,Z 107,A 12.2133,B 24.9335,C -1.8832,E1 25.1531,E2 433.4053} C_DIS
LIN {X 102.3868,Y 33.2288,Z 107,A 13.9151,B 24.9329,C -1.8925,E1 25.1516,E2 431.6913} C_DIS
LIN {X 101.1692,Y 36.7695,Z 107,A 15.7713,B 24.9329,C -1.8925,E1 25.1499,E2 429.8456} C_DIS
LIN {X 100.2053,Y 39.3204,Z 107,A 17.252,B 24.9325,C -1.898,E1 25.1484,E2 428.3601} C_DIS
LIN {X 99.0536,Y 42.1391,Z 107,A 18.9696,B 24.9318,C -1.9069,E1 25.1466,E2 426.6309} C_DIS
LIN {X 97.8781,Y 44.8049,Z 107,A 20.6667,B 24.9311,C -1.9177,E1 25.1446,E2 424.9174} C_DIS
Enddeposition()
END
